gfCNCPoint6[10875] = {X 516.8418, Y 19.7797, Z -8.0000, A 0.000, B 0.000, C 0.000 }
gfCNCPoint6[10876] = {X 516.3652, Y 19.0212, Z -8.0000, A 0.000, B 0.000, C 0.000 }
gfCNCPoint6[10877] = {X 516.0694, Y 18.1758, Z -8.0000, A 0.000, B 0.000, C 0.000 }
gfCNCPoint6[10878] = {X 515.9691, Y 17.2857, Z -8.0000, A 0.000, B 0.000, C 0.000 }
gfCNCPoint6[10879] = {X 515.9691, Y 10.3077, Z -8.0000, A 0.000, B 0.000, C 0.000 }
gfCNCPoint6[10880] = {X 516.0694, Y 9.4176, Z -8.0000, A 0.000, B 0.000, C 0.000 }
gfCNCPoint6[10881] = {X 516.3652, Y 8.5721, Z -8.0000, A 0.000, B 0.000, C 0.000 }
gfCNCPoint6[10882] = {X 516.8418, Y 7.8137, Z -8.0000, A 0.000, B 0.000, C 0.000 }
gfCNCPoint6[10883] = {X 517.4752, Y 7.1803, Z -8.0000, A 0.000, B 0.000, C 0.000 }
gfCNCPoint6[10884] = {X 518.2336, Y 6.7038, Z -8.0000, A 0.000, B 0.000, C 0.000 }
gfCNCPoint6[10885] = {X 519.0791, Y 6.4080, Z -8.0000, A 0.000, B 0.000, C 0.000 }
gfCNCPoint6[10886] = {X 519.9692, Y 6.3077, Z -8.0000, A 0.000, B 0.000, C 0.000 }
gfCNCPoint6[10887] = {X 520.6473, Y 6.3079, Z -8.0000, A 0.000, B 0.000, C 0.000 }
gfCNCPoint6[10888] = {X 521.4439, Y 6.3954, Z -8.0000, A 0.000, B 0.000, C 0.000 }
gfCNCPoint6[10889] = {X 522.2072, Y 6.6401, Z -8.0000, A 0.000, B 0.000, C 0.000 }
gfCNCPoint6[10890] = {X 522.9063, Y 7.0319, Z -8.0000, A 0.000, B 0.000, C 0.000 }
gfCNCPoint6[10891] = {X 523.5133, Y 7.5553, Z -8.0000, A 0.000, B 0.000, C 0.000 }
gfCNCPoint6[10892] = {X 524.0037, Y 8.1892, Z -8.0000, A 0.000, B 0.000, C 0.000 }
gfCNCPoint6[10893] = {X 533.9633, Y 8.1892, Z -8.0000, A 0.000, B 0.000, C 0.000 }
gfCNCPoint6[10894] = {X 533.9633, Y 4.1092, Z -8.0000, A 0.000, B 0.000, C 0.000 }
gfCNCPoint6[10895] = {X 533.9633, Y 4.1092, Z -5.0000, A 0.000, B 0.000, C 0.000 }
gfCNCPoint6[10896] = {X 533.9633, Y 4.1092, Z 11.0000, A 0.000, B 0.000, C 0.000 }
gfCNCPoint6[10897] = {X 419.6152, Y 26.5282, Z 11.0000, A 0.000, B 0.000, C 0.000 }
gfCNCPoint6[10898] = {X 419.6152, Y 26.5282, Z -5.0000, A 0.000, B 0.000, C 0.000 }
gfCNCPoint6[10899] = {X 419.6152, Y 26.5282, Z -8.0000, A 0.000, B 0.000, C 0.000 }
gfCNCPoint6[10900] = {X 416.1517, Y 24.3717, Z -8.0000, A 0.000, B 0.000, C 0.000 }
gfCNCPoint6[10901] = {X 411.5482, Y 31.7655, Z -8.0000, A 0.000, B 0.000, C 0.000 }
gfCNCPoint6[10902] = {X 411.5488, Y 40.8974, Z -8.0000, A 0.000, B 0.000, C 0.000 }
gfCNCPoint6[10903] = {X 412.1870, Y 41.5833, Z -8.0000, A 0.000, B 0.000, C 0.000 }
gfCNCPoint6[10904] = {X 412.6670, Y 42.3878, Z -8.0000, A 0.000, B 0.000, C 0.000 }
gfCNCPoint6[10905] = {X 412.9674, Y 43.2752, Z -8.0000, A 0.000, B 0.000, C 0.000 }
gfCNCPoint6[10906] = {X 413.0747, Y 44.2059, Z -8.0000, A 0.000, B 0.000, C 0.000 }
gfCNCPoint6[10907] = {X 413.0745, Y 45.0415, Z -8.0000, A 0.000, B 0.000, C 0.000 }
gfCNCPoint6[10908] = {X 412.9583, Y 45.9960, Z -8.0000, A 0.000, B 0.000, C 0.000 }
gfCNCPoint6[10909] = {X 412.6339, Y 46.9011, Z -8.0000, A 0.000, B 0.000, C 0.000 }
gfCNCPoint6[10910] = {X 412.1173, Y 47.7120, Z -8.0000, A 0.000, B 0.000, C 0.000 }
gfCNCPoint6[10911] = {X 411.4342, Y 48.3886, Z -8.0000, A 0.000, B 0.000, C 0.000 }
gfCNCPoint6[10912] = {X 410.6184, Y 48.8973, Z -8.0000, A 0.000, B 0.000, C 0.000 }
gfCNCPoint6[10913] = {X 409.7102, Y 49.2130, Z -8.0000, A 0.000, B 0.000, C 0.000 }
gfCNCPoint6[10914] = {X 408.7547, Y 49.3200, Z -8.0000, A 0.000, B 0.000, C 0.000 }
gfCNCPoint6[10915] = {X 402.3112, Y 49.3200, Z -8.0000, A 0.000, B 0.000, C 0.000 }
gfCNCPoint6[10916] = {X 401.3546, Y 49.2127, Z -8.0000, A 0.000, B 0.000, C 0.000 }
gfCNCPoint6[10917] = {X 400.4455, Y 48.8963, Z -8.0000, A 0.000, B 0.000, C 0.000 }
gfCNCPoint6[10918] = {X 399.6290, Y 48.3864, Z -8.0000, A 0.000, B 0.000, C 0.000 }
gfCNCPoint6[10919] = {X 398.9457, Y 47.7084, Z -8.0000, A 0.000, B 0.000, C 0.000 }
gfCNCPoint6[10920] = {X 398.4295, Y 46.8959, Z -8.0000, A 0.000, B 0.000, C 0.000 }
gfCNCPoint6[10921] = {X 398.1060, Y 45.9892, Z -8.0000, A 0.000, B 0.000, C 0.000 }
gfCNCPoint6[10922] = {X 397.9913, Y 45.0335, Z -8.0000, A 0.000, B 0.000, C 0.000 }
gfCNCPoint6[10923] = {X 397.9916, Y 44.1528, Z -8.0000, A 0.000, B 0.000, C 0.000 }
gfCNCPoint6[10924] = {X 398.1015, Y 43.2391, Z -8.0000, A 0.000, B 0.000, C 0.000 }
gfCNCPoint6[10925] = {X 398.4024, Y 42.3694, Z -8.0000, A 0.000, B 0.000, C 0.000 }
gfCNCPoint6[10926] = {X 398.8807, Y 41.5832, Z -8.0000, A 0.000, B 0.000, C 0.000 }
gfCNCPoint6[10927] = {X 399.5147, Y 40.9161, Z -8.0000, A 0.000, B 0.000, C 0.000 }
gfCNCPoint6[10928] = {X 399.4729, Y 31.6029, Z -8.0000, A 0.000, B 0.000, C 0.000 }
gfCNCPoint6[10929] = {X 393.4346, Y 21.1023, Z -8.0000, A 0.000, B 0.000, C 0.000 }
gfCNCPoint6[10930] = {X 392.5863, Y 19.6607, Z -8.0000, A 0.000, B 0.000, C 0.000 }
gfCNCPoint6[10931] = {X 391.7093, Y 18.2363, Z -8.0000, A 0.000, B 0.000, C 0.000 }
gfCNCPoint6[10932] = {X 391.2277, Y 17.5680, Z -8.0000, A 0.000, B 0.000, C 0.000 }
gfCNCPoint6[10933] = {X 390.6666, Y 16.9651, Z -8.0000, A 0.000, B 0.000, C 0.000 }
gfCNCPoint6[10934] = {X 389.7900, Y 16.4727, Z -8.0000, A 0.000, B 0.000, C 0.000 }
gfCNCPoint6[10935] = {X 389.0509, Y 15.7909, Z -8.0000, A 0.000, B 0.000, C 0.000 }
gfCNCPoint6[10936] = {X 388.4895, Y 14.9568, Z -8.0000, A 0.000, B 0.000, C 0.000 }
gfCNCPoint6[10937] = {X 388.1361, Y 14.0155, Z -8.0000, A 0.000, B 0.000, C 0.000 }
gfCNCPoint6[10938] = {X 388.0098, Y 13.0180, Z -8.0000, A 0.000, B 0.000, C 0.000 }
gfCNCPoint6[10939] = {X 388.0096, Y 12.1868, Z -8.0000, A 0.000, B 0.000, C 0.000 }
gfCNCPoint6[10940] = {X 388.1179, Y 11.2255, Z -8.0000, A 0.000, B 0.000, C 0.000 }
gfCNCPoint6[10941] = {X 388.4374, Y 10.3125, Z -8.0000, A 0.000, B 0.000, C 0.000 }
gfCNCPoint6[10942] = {X 388.9521, Y 9.4933, Z -8.0000, A 0.000, B 0.000, C 0.000 }
gfCNCPoint6[10943] = {X 389.6361, Y 8.8093, Z -8.0000, A 0.000, B 0.000, C 0.000 }
gfCNCPoint6[10944] = {X 390.4552, Y 8.2946, Z -8.0000, A 0.000, B 0.000, C 0.000 }
gfCNCPoint6[10945] = {X 391.3683, Y 7.9751, Z -8.0000, A 0.000, B 0.000, C 0.000 }
gfCNCPoint6[10946] = {X 392.3296, Y 7.8668, Z -8.0000, A 0.000, B 0.000, C 0.000 }
gfCNCPoint6[10947] = {X 399.1118, Y 7.8668, Z -8.0000, A 0.000, B 0.000, C 0.000 }
gfCNCPoint6[10948] = {X 400.0730, Y 7.9751, Z -8.0000, A 0.000, B 0.000, C 0.000 }
gfCNCPoint6[10949] = {X 400.9861, Y 8.2946, Z -8.0000, A 0.000, B 0.000, C 0.000 }
gfCNCPoint6[10950] = {X 401.8052, Y 8.8093, Z -8.0000, A 0.000, B 0.000, C 0.000 }
gfCNCPoint6[10951] = {X 402.4893, Y 9.4933, Z -8.0000, A 0.000, B 0.000, C 0.000 }
gfCNCPoint6[10952] = {X 403.0039, Y 10.3124, Z -8.0000, A 0.000, B 0.000, C 0.000 }
gfCNCPoint6[10953] = {X 403.3234, Y 11.2255, Z -8.0000, A 0.000, B 0.000, C 0.000 }
gfCNCPoint6[10954] = {X 403.4318, Y 12.1868, Z -8.0000, A 0.000, B 0.000, C 0.000 }
gfCNCPoint6[10955] = {X 403.4318, Y 12.9782, Z -8.0000, A 0.000, B 0.000, C 0.000 }
gfCNCPoint6[10956] = {X 403.3293, Y 13.9135, Z -8.0000, A 0.000, B 0.000, C 0.000 }
gfCNCPoint6[10957] = {X 403.0267, Y 14.8044, Z -8.0000, A 0.000, B 0.000, C 0.000 }
gfCNCPoint6[10958] = {X 405.3554, Y 18.8222, Z -8.0000, A 0.000, B 0.000, C 0.000 }
gfCNCPoint6[10959] = {X 407.8730, Y 14.7530, Z -8.0000, A 0.000, B 0.000, C 0.000 }
gfCNCPoint6[10960] = {X 407.5919, Y 13.9039, Z -8.0000, A 0.000, B 0.000, C 0.000 }
gfCNCPoint6[10961] = {X 407.4917, Y 13.0151, Z -8.0000, A 0.000, B 0.000, C 0.000 }
gfCNCPoint6[10962] = {X 407.4915, Y 12.1868, Z -8.0000, A 0.000, B 0.000, C 0.000 }
gfCNCPoint6[10963] = {X 407.5999, Y 11.2255, Z -8.0000, A 0.000, B 0.000, C 0.000 }
gfCNCPoint6[10964] = {X 407.9194, Y 10.3124, Z -8.0000, A 0.000, B 0.000, C 0.000 }
gfCNCPoint6[10965] = {X 408.4340, Y 9.4933, Z -8.0000, A 0.000, B 0.000, C 0.000 }
gfCNCPoint6[10966] = {X 409.1181, Y 8.8093, Z -8.0000, A 0.000, B 0.000, C 0.000 }
gfCNCPoint6[10967] = {X 409.9372, Y 8.2946, Z -8.0000, A 0.000, B 0.000, C 0.000 }
gfCNCPoint6[10968] = {X 410.8502, Y 7.9751, Z -8.0000, A 0.000, B 0.000, C 0.000 }
gfCNCPoint6[10969] = {X 411.8115, Y 7.8668, Z -8.0000, A 0.000, B 0.000, C 0.000 }
gfCNCPoint6[10970] = {X 419.3245, Y 7.8668, Z -8.0000, A 0.000, B 0.000, C 0.000 }
gfCNCPoint6[10971] = {X 420.2858, Y 7.9751, Z -8.0000, A 0.000, B 0.000, C 0.000 }
gfCNCPoint6[10972] = {X 421.1988, Y 8.2946, Z -8.0000, A 0.000, B 0.000, C 0.000 }
gfCNCPoint6[10973] = {X 422.0179, Y 8.8093, Z -8.0000, A 0.000, B 0.000, C 0.000 }
gfCNCPoint6[10974] = {X 422.7020, Y 9.4933, Z -8.0000, A 0.000, B 0.000, C 0.000 }
gfCNCPoint6[10975] = {X 423.2166, Y 10.3124, Z -8.0000, A 0.000, B 0.000, C 0.000 }
gfCNCPoint6[10976] = {X 423.5361, Y 11.2255, Z -8.0000, A 0.000, B 0.000, C 0.000 }
gfCNCPoint6[10977] = {X 423.6445, Y 12.1868, Z -8.0000, A 0.000, B 0.000, C 0.000 }
gfCNCPoint6[10978] = {X 423.6445, Y 12.9801, Z -8.0000, A 0.000, B 0.000, C 0.000 }
gfCNCPoint6[10979] = {X 423.5522, Y 13.8467, Z -8.0000, A 0.000, B 0.000, C 0.000 }
gfCNCPoint6[10980] = {X 423.2901, Y 14.6779, Z -8.0000, A 0.000, B 0.000, C 0.000 }
gfCNCPoint6[10981] = {X 422.8686, Y 15.4407, Z -8.0000, A 0.000, B 0.000, C 0.000 }
gfCNCPoint6[10982] = {X 422.3045, Y 16.1050, Z -8.0000, A 0.000, B 0.000, C 0.000 }
gfCNCPoint6[10983] = {X 421.6199, Y 16.6444, Z -8.0000, A 0.000, B 0.000, C 0.000 }
gfCNCPoint6[10984] = {X 420.8421, Y 17.0376, Z -8.0000, A 0.000, B 0.000, C 0.000 }
gfCNCPoint6[10985] = {X 420.1257, Y 18.0009, Z -8.0000, A 0.000, B 0.000, C 0.000 }
gfCNCPoint6[10986] = {X 419.4776, Y 19.0115, Z -8.0000, A 0.000, B 0.000, C 0.000 }
gfCNCPoint6[10987] = {X 417.9942, Y 21.4124, Z -8.0000, A 0.000, B 0.000, C 0.000 }
gfCNCPoint6[10988] = {X 416.1517, Y 24.3717, Z -8.0000, A 0.000, B 0.000, C 0.000 }
gfCNCPoint6[10989] = {X 419.5473, Y 26.4859, Z -8.0000, A 0.000, B 0.000, C 0.000 }
gfCNCPoint6[10990] = {X 416.0838, Y 24.3294, Z -8.0000, A 0.000, B 0.000, C 0.000 }
gfCNCPoint6[10991] = {X 411.4682, Y 31.7426, Z -8.0000, A 0.000, B 0.000, C 0.000 }
gfCNCPoint6[10992] = {X 411.4688, Y 40.9341, Z -8.0000, A 0.000, B 0.000, C 0.000 }
gfCNCPoint6[10993] = {X 412.1066, Y 41.6095, Z -8.0000, A 0.000, B 0.000, C 0.000 }
gfCNCPoint6[10994] = {X 412.5867, Y 42.4049, Z -8.0000, A 0.000, B 0.000, C 0.000 }
gfCNCPoint6[10995] = {X 412.8873, Y 43.2839, Z -8.0000, A 0.000, B 0.000, C 0.000 }
gfCNCPoint6[10996] = {X 412.9947, Y 44.2067, Z -8.0000, A 0.000, B 0.000, C 0.000 }
gfCNCPoint6[10997] = {X 412.9945, Y 45.0408, Z -8.0000, A 0.000, B 0.000, C 0.000 }
gfCNCPoint6[10998] = {X 412.8805, Y 45.9775, Z -8.0000, A 0.000, B 0.000, C 0.000 }
gfCNCPoint6[10999] = {X 412.5621, Y 46.8659, Z -8.0000, A 0.000, B 0.000, C 0.000 }
gfCNCPoint6[11000] = {X 412.0551, Y 47.6618, Z -8.0000, A 0.000, B 0.000, C 0.000 }
gfCNCPoint6[11001] = {X 411.3846, Y 48.3258, Z -8.0000, A 0.000, B 0.000, C 0.000 }
gfCNCPoint6[11002] = {X 410.5838, Y 48.8251, Z -8.0000, A 0.000, B 0.000, C 0.000 }
gfCNCPoint6[11003] = {X 409.6925, Y 49.1350, Z -8.0000, A 0.000, B 0.000, C 0.000 }
gfCNCPoint6[11004] = {X 408.7547, Y 49.2400, Z -8.0000, A 0.000, B 0.000, C 0.000 }
gfCNCPoint6[11005] = {X 402.3112, Y 49.2400, Z -8.0000, A 0.000, B 0.000, C 0.000 }
gfCNCPoint6[11006] = {X 401.3723, Y 49.1347, Z -8.0000, A 0.000, B 0.000, C 0.000 }
gfCNCPoint6[11007] = {X 400.4800, Y 48.8242, Z -8.0000, A 0.000, B 0.000, C 0.000 }
gfCNCPoint6[11008] = {X 399.6786, Y 48.3237, Z -8.0000, A 0.000, B 0.000, C 0.000 }
gfCNCPoint6[11009] = {X 399.0080, Y 47.6582, Z -8.0000, A 0.000, B 0.000, C 0.000 }
gfCNCPoint6[11010] = {X 398.5013, Y 46.8608, Z -8.0000, A 0.000, B 0.000, C 0.000 }
gfCNCPoint6[11011] = {X 398.1839, Y 45.9709, Z -8.0000, A 0.000, B 0.000, C 0.000 }
gfCNCPoint6[11012] = {X 398.0713, Y 45.0329, Z -8.0000, A 0.000, B 0.000, C 0.000 }
gfCNCPoint6[11013] = {X 398.0716, Y 44.1538, Z -8.0000, A 0.000, B 0.000, C 0.000 }
gfCNCPoint6[11014] = {X 398.1815, Y 43.2480, Z -8.0000, A 0.000, B 0.000, C 0.000 }
gfCNCPoint6[11015] = {X 398.4827, Y 42.3867, Z -8.0000, A 0.000, B 0.000, C 0.000 }
gfCNCPoint6[11016] = {X 398.9612, Y 41.6098, Z -8.0000, A 0.000, B 0.000, C 0.000 }
gfCNCPoint6[11017] = {X 399.5948, Y 40.9532, Z -8.0000, A 0.000, B 0.000, C 0.000 }
gfCNCPoint6[11018] = {X 399.5528, Y 31.5814, Z -8.0000, A 0.000, B 0.000, C 0.000 }
gfCNCPoint6[11019] = {X 393.5040, Y 21.0625, Z -8.0000, A 0.000, B 0.000, C 0.000 }
gfCNCPoint6[11020] = {X 392.6548, Y 19.6194, Z -8.0000, A 0.000, B 0.000, C 0.000 }
gfCNCPoint6[11021] = {X 391.7770, Y 18.1936, Z -8.0000, A 0.000, B 0.000, C 0.000 }
gfCNCPoint6[11022] = {X 391.2849, Y 17.5116, Z -8.0000, A 0.000, B 0.000, C 0.000 }
gfCNCPoint6[11023] = {X 390.7109, Y 16.8969, Z -8.0000, A 0.000, B 0.000, C 0.000 }
gfCNCPoint6[11024] = {X 389.8465, Y 16.4148, Z -8.0000, A 0.000, B 0.000, C 0.000 }
gfCNCPoint6[11025] = {X 389.1174, Y 15.7455, Z -8.0000, A 0.000, B 0.000, C 0.000 }
gfCNCPoint6[11026] = {X 388.5633, Y 14.9254, Z -8.0000, A 0.000, B 0.000, C 0.000 }
gfCNCPoint6[11027] = {X 388.2144, Y 13.9992, Z -8.0000, A 0.000, B 0.000, C 0.000 }
gfCNCPoint6[11028] = {X 388.0898, Y 13.0173, Z -8.0000, A 0.000, B 0.000, C 0.000 }
gfCNCPoint6[11029] = {X 388.0896, Y 12.1868, Z -8.0000, A 0.000, B 0.000, C 0.000 }
gfCNCPoint6[11030] = {X 388.1959, Y 11.2433, Z -8.0000, A 0.000, B 0.000, C 0.000 }
gfCNCPoint6[11031] = {X 388.5095, Y 10.3472, Z -8.0000, A 0.000, B 0.000, C 0.000 }
gfCNCPoint6[11032] = {X 389.0147, Y 9.5432, Z -8.0000, A 0.000, B 0.000, C 0.000 }
gfCNCPoint6[11033] = {X 389.6860, Y 8.8719, Z -8.0000, A 0.000, B 0.000, C 0.000 }
gfCNCPoint6[11034] = {X 390.4900, Y 8.3667, Z -8.0000, A 0.000, B 0.000, C 0.000 }
gfCNCPoint6[11035] = {X 391.3861, Y 8.0531, Z -8.0000, A 0.000, B 0.000, C 0.000 }
gfCNCPoint6[11036] = {X 392.3296, Y 7.9468, Z -8.0000, A 0.000, B 0.000, C 0.000 }
gfCNCPoint6[11037] = {X 399.1118, Y 7.9468, Z -8.0000, A 0.000, B 0.000, C 0.000 }
gfCNCPoint6[11038] = {X 400.0552, Y 8.0531, Z -8.0000, A 0.000, B 0.000, C 0.000 }
gfCNCPoint6[11039] = {X 400.9514, Y 8.3667, Z -8.0000, A 0.000, B 0.000, C 0.000 }
gfCNCPoint6[11040] = {X 401.7554, Y 8.8718, Z -8.0000, A 0.000, B 0.000, C 0.000 }
gfCNCPoint6[11041] = {X 402.4267, Y 9.5432, Z -8.0000, A 0.000, B 0.000, C 0.000 }
gfCNCPoint6[11042] = {X 402.9319, Y 10.3471, Z -8.0000, A 0.000, B 0.000, C 0.000 }
gfCNCPoint6[11043] = {X 403.2455, Y 11.2433, Z -8.0000, A 0.000, B 0.000, C 0.000 }
gfCNCPoint6[11044] = {X 403.3518, Y 12.1868, Z -8.0000, A 0.000, B 0.000, C 0.000 }
gfCNCPoint6[11045] = {X 403.3518, Y 12.9782, Z -8.0000, A 0.000, B 0.000, C 0.000 }
gfCNCPoint6[11046] = {X 403.2466, Y 13.9164, Z -8.0000, A 0.000, B 0.000, C 0.000 }
gfCNCPoint6[11047] = {X 402.9364, Y 14.8081, Z -8.0000, A 0.000, B 0.000, C 0.000 }
gfCNCPoint6[11048] = {X 405.3532, Y 18.9779, Z -8.0000, A 0.000, B 0.000, C 0.000 }
gfCNCPoint6[11049] = {X 407.9636, Y 14.7587, Z -8.0000, A 0.000, B 0.000, C 0.000 }
gfCNCPoint6[11050] = {X 407.6747, Y 13.9075, Z -8.0000, A 0.000, B 0.000, C 0.000 }
gfCNCPoint6[11051] = {X 407.5717, Y 13.0144, Z -8.0000, A 0.000, B 0.000, C 0.000 }
gfCNCPoint6[11052] = {X 407.5715, Y 12.1868, Z -8.0000, A 0.000, B 0.000, C 0.000 }
gfCNCPoint6[11053] = {X 407.6778, Y 11.2433, Z -8.0000, A 0.000, B 0.000, C 0.000 }
gfCNCPoint6[11054] = {X 407.9914, Y 10.3471, Z -8.0000, A 0.000, B 0.000, C 0.000 }
gfCNCPoint6[11055] = {X 408.4966, Y 9.5432, Z -8.0000, A 0.000, B 0.000, C 0.000 }
gfCNCPoint6[11056] = {X 409.1679, Y 8.8718, Z -8.0000, A 0.000, B 0.000, C 0.000 }
gfCNCPoint6[11057] = {X 409.9719, Y 8.3667, Z -8.0000, A 0.000, B 0.000, C 0.000 }
gfCNCPoint6[11058] = {X 410.8681, Y 8.0531, Z -8.0000, A 0.000, B 0.000, C 0.000 }
gfCNCPoint6[11059] = {X 411.8115, Y 7.9468, Z -8.0000, A 0.000, B 0.000, C 0.000 }
gfCNCPoint6[11060] = {X 419.3245, Y 7.9468, Z -8.0000, A 0.000, B 0.000, C 0.000 }
gfCNCPoint6[11061] = {X 420.2679, Y 8.0531, Z -8.0000, A 0.000, B 0.000, C 0.000 }
gfCNCPoint6[11062] = {X 421.1641, Y 8.3667, Z -8.0000, A 0.000, B 0.000, C 0.000 }
gfCNCPoint6[11063] = {X 421.9681, Y 8.8718, Z -8.0000, A 0.000, B 0.000, C 0.000 }
gfCNCPoint6[11064] = {X 422.6394, Y 9.5432, Z -8.0000, A 0.000, B 0.000, C 0.000 }
gfCNCPoint6[11065] = {X 423.1446, Y 10.3471, Z -8.0000, A 0.000, B 0.000, C 0.000 }
gfCNCPoint6[11066] = {X 423.4582, Y 11.2433, Z -8.0000, A 0.000, B 0.000, C 0.000 }
gfCNCPoint6[11067] = {X 423.5645, Y 12.1868, Z -8.0000, A 0.000, B 0.000, C 0.000 }
gfCNCPoint6[11068] = {X 423.5645, Y 12.9795, Z -8.0000, A 0.000, B 0.000, C 0.000 }
gfCNCPoint6[11069] = {X 423.4731, Y 13.8339, Z -8.0000, A 0.000, B 0.000, C 0.000 }
gfCNCPoint6[11070] = {X 423.2137, Y 14.6529, Z -8.0000, A 0.000, B 0.000, C 0.000 }
gfCNCPoint6[11071] = {X 422.7967, Y 15.4041, Z -8.0000, A 0.000, B 0.000, C 0.000 }
gfCNCPoint6[11072] = {X 422.2386, Y 16.0574, Z -8.0000, A 0.000, B 0.000, C 0.000 }
gfCNCPoint6[11073] = {X 421.5618, Y 16.5866, Z -8.0000, A 0.000, B 0.000, C 0.000 }
gfCNCPoint6[11074] = {X 420.7932, Y 16.9707, Z -8.0000, A 0.000, B 0.000, C 0.000 }
gfCNCPoint6[11075] = {X 420.0662, Y 17.9462, Z -8.0000, A 0.000, B 0.000, C 0.000 }
gfCNCPoint6[11076] = {X 419.4091, Y 18.9700, Z -8.0000, A 0.000, B 0.000, C 0.000 }
gfCNCPoint6[11077] = {X 417.9262, Y 21.3702, Z -8.0000, A 0.000, B 0.000, C 0.000 }
gfCNCPoint6[11078] = {X 416.0838, Y 24.3294, Z -8.0000, A 0.000, B 0.000, C 0.000 }
gfCNCPoint6[11079] = {X 419.4794, Y 26.4436, Z -8.0000, A 0.000, B 0.000, C 0.000 }
gfCNCPoint6[11080] = {X 416.0159, Y 24.2871, Z -8.0000, A 0.000, B 0.000, C 0.000 }
gfCNCPoint6[11081] = {X 411.3882, Y 31.7197, Z -8.0000, A 0.000, B 0.000, C 0.000 }
gfCNCPoint6[11082] = {X 411.3888, Y 40.9711, Z -8.0000, A 0.000, B 0.000, C 0.000 }
gfCNCPoint6[11083] = {X 412.0262, Y 41.6361, Z -8.0000, A 0.000, B 0.000, C 0.000 }
gfCNCPoint6[11084] = {X 412.5064, Y 42.4220, Z -8.0000, A 0.000, B 0.000, C 0.000 }
gfCNCPoint6[11085] = {X 412.8072, Y 43.2926, Z -8.0000, A 0.000, B 0.000, C 0.000 }
gfCNCPoint6[11086] = {X 412.9147, Y 44.2074, Z -8.0000, A 0.000, B 0.000, C 0.000 }
gfCNCPoint6[11087] = {X 412.9145, Y 45.0400, Z -8.0000, A 0.000, B 0.000, C 0.000 }
gfCNCPoint6[11088] = {X 412.8026, Y 45.9591, Z -8.0000, A 0.000, B 0.000, C 0.000 }
gfCNCPoint6[11089] = {X 412.4902, Y 46.8306, Z -8.0000, A 0.000, B 0.000, C 0.000 }
gfCNCPoint6[11090] = {X 411.9928, Y 47.6115, Z -8.0000, A 0.000, B 0.000, C 0.000 }
gfCNCPoint6[11091] = {X 411.3350, Y 48.2631, Z -8.0000, A 0.000, B 0.000, C 0.000 }
gfCNCPoint6[11092] = {X 410.5493, Y 48.7530, Z -8.0000, A 0.000, B 0.000, C 0.000 }
gfCNCPoint6[11093] = {X 409.6748, Y 49.0570, Z -8.0000, A 0.000, B 0.000, C 0.000 }
gfCNCPoint6[11094] = {X 408.7547, Y 49.1600, Z -8.0000, A 0.000, B 0.000, C 0.000 }
gfCNCPoint6[11095] = {X 402.3112, Y 49.1600, Z -8.0000, A 0.000, B 0.000, C 0.000 }
gfCNCPoint6[11096] = {X 401.3900, Y 49.0567, Z -8.0000, A 0.000, B 0.000, C 0.000 }
gfCNCPoint6[11097] = {X 400.5146, Y 48.7520, Z -8.0000, A 0.000, B 0.000, C 0.000 }
gfCNCPoint6[11098] = {X 399.7283, Y 48.2610, Z -8.0000, A 0.000, B 0.000, C 0.000 }
gfCNCPoint6[11099] = {X 399.0703, Y 47.6081, Z -8.0000, A 0.000, B 0.000, C 0.000 }
gfCNCPoint6[11100] = {X 398.5732, Y 46.8257, Z -8.0000, A 0.000, B 0.000, C 0.000 }
gfCNCPoint6[11101] = {X 398.2617, Y 45.9526, Z -8.0000, A 0.000, B 0.000, C 0.000 }
gfCNCPoint6[11102] = {X 398.1513, Y 45.0322, Z -8.0000, A 0.000, B 0.000, C 0.000 }
gfCNCPoint6[11103] = {X 398.1516, Y 44.1549, Z -8.0000, A 0.000, B 0.000, C 0.000 }
gfCNCPoint6[11104] = {X 398.2616, Y 43.2570, Z -8.0000, A 0.000, B 0.000, C 0.000 }
gfCNCPoint6[11105] = {X 398.5630, Y 42.4041, Z -8.0000, A 0.000, B 0.000, C 0.000 }
gfCNCPoint6[11106] = {X 399.0417, Y 41.6366, Z -8.0000, A 0.000, B 0.000, C 0.000 }
gfCNCPoint6[11107] = {X 399.6750, Y 40.9907, Z -8.0000, A 0.000, B 0.000, C 0.000 }
gfCNCPoint6[11108] = {X 399.6327, Y 31.5599, Z -8.0000, A 0.000, B 0.000, C 0.000 }
gfCNCPoint6[11109] = {X 393.5733, Y 21.0226, Z -8.0000, A 0.000, B 0.000, C 0.000 }
gfCNCPoint6[11110] = {X 392.7234, Y 19.5782, Z -8.0000, A 0.000, B 0.000, C 0.000 }
gfCNCPoint6[11111] = {X 391.8447, Y 18.1510, Z -8.0000, A 0.000, B 0.000, C 0.000 }
gfCNCPoint6[11112] = {X 391.3420, Y 17.4550, Z -8.0000, A 0.000, B 0.000, C 0.000 }
gfCNCPoint6[11113] = {X 390.7550, Y 16.8285, Z -8.0000, A 0.000, B 0.000, C 0.000 }
gfCNCPoint6[11114] = {X 389.9028, Y 16.3568, Z -8.0000, A 0.000, B 0.000, C 0.000 }
gfCNCPoint6[11115] = {X 389.1837, Y 15.6999, Z -8.0000, A 0.000, B 0.000, C 0.000 }
gfCNCPoint6[11116] = {X 388.6370, Y 14.8938, Z -8.0000, A 0.000, B 0.000, C 0.000 }
gfCNCPoint6[11117] = {X 388.2928, Y 13.9827, Z -8.0000, A 0.000, B 0.000, C 0.000 }
gfCNCPoint6[11118] = {X 388.1698, Y 13.0166, Z -8.0000, A 0.000, B 0.000, C 0.000 }
gfCNCPoint6[11119] = {X 388.1696, Y 12.1868, Z -8.0000, A 0.000, B 0.000, C 0.000 }
gfCNCPoint6[11120] = {X 388.2739, Y 11.2611, Z -8.0000, A 0.000, B 0.000, C 0.000 }
gfCNCPoint6[11121] = {X 388.5816, Y 10.3819, Z -8.0000, A 0.000, B 0.000, C 0.000 }
gfCNCPoint6[11122] = {X 389.0772, Y 9.5931, Z -8.0000, A 0.000, B 0.000, C 0.000 }
gfCNCPoint6[11123] = {X 389.7359, Y 8.9344, Z -8.0000, A 0.000, B 0.000, C 0.000 }
gfCNCPoint6[11124] = {X 390.5247, Y 8.4388, Z -8.0000, A 0.000, B 0.000, C 0.000 }
gfCNCPoint6[11125] = {X 391.4039, Y 8.1311, Z -8.0000, A 0.000, B 0.000, C 0.000 }
gfCNCPoint6[11126] = {X 392.3296, Y 8.0268, Z -8.0000, A 0.000, B 0.000, C 0.000 }
gfCNCPoint6[11127] = {X 399.1118, Y 8.0268, Z -8.0000, A 0.000, B 0.000, C 0.000 }
gfCNCPoint6[11128] = {X 400.0374, Y 8.1311, Z -8.0000, A 0.000, B 0.000, C 0.000 }
gfCNCPoint6[11129] = {X 400.9167, Y 8.4388, Z -8.0000, A 0.000, B 0.000, C 0.000 }
gfCNCPoint6[11130] = {X 401.7055, Y 8.9344, Z -8.0000, A 0.000, B 0.000, C 0.000 }
gfCNCPoint6[11131] = {X 402.3642, Y 9.5931, Z -8.0000, A 0.000, B 0.000, C 0.000 }
gfCNCPoint6[11132] = {X 402.8598, Y 10.3819, Z -8.0000, A 0.000, B 0.000, C 0.000 }
gfCNCPoint6[11133] = {X 403.1675, Y 11.2611, Z -8.0000, A 0.000, B 0.000, C 0.000 }
gfCNCPoint6[11134] = {X 403.2718, Y 12.1868, Z -8.0000, A 0.000, B 0.000, C 0.000 }
gfCNCPoint6[11135] = {X 403.2718, Y 12.9782, Z -8.0000, A 0.000, B 0.000, C 0.000 }
gfCNCPoint6[11136] = {X 403.1639, Y 13.9192, Z -8.0000, A 0.000, B 0.000, C 0.000 }
gfCNCPoint6[11137] = {X 402.8459, Y 14.8115, Z -8.0000, A 0.000, B 0.000, C 0.000 }
gfCNCPoint6[11138] = {X 405.3509, Y 19.1335, Z -8.0000, A 0.000, B 0.000, C 0.000 }
gfCNCPoint6[11139] = {X 408.0544, Y 14.7640, Z -8.0000, A 0.000, B 0.000, C 0.000 }
gfCNCPoint6[11140] = {X 407.7575, Y 13.9109, Z -8.0000, A 0.000, B 0.000, C 0.000 }
gfCNCPoint6[11141] = {X 407.6517, Y 13.0137, Z -8.0000, A 0.000, B 0.000, C 0.000 }
gfCNCPoint6[11142] = {X 407.6515, Y 12.1868, Z -8.0000, A 0.000, B 0.000, C 0.000 }
gfCNCPoint6[11143] = {X 407.7558, Y 11.2611, Z -8.0000, A 0.000, B 0.000, C 0.000 }
gfCNCPoint6[11144] = {X 408.0635, Y 10.3819, Z -8.0000, A 0.000, B 0.000, C 0.000 }
gfCNCPoint6[11145] = {X 408.5591, Y 9.5931, Z -8.0000, A 0.000, B 0.000, C 0.000 }
gfCNCPoint6[11146] = {X 409.2178, Y 8.9344, Z -8.0000, A 0.000, B 0.000, C 0.000 }
gfCNCPoint6[11147] = {X 410.0066, Y 8.4388, Z -8.0000, A 0.000, B 0.000, C 0.000 }
gfCNCPoint6[11148] = {X 410.8859, Y 8.1311, Z -8.0000, A 0.000, B 0.000, C 0.000 }
gfCNCPoint6[11149] = {X 411.8115, Y 8.0268, Z -8.0000, A 0.000, B 0.000, C 0.000 }
gfCNCPoint6[11150] = {X 419.3245, Y 8.0268, Z -8.0000, A 0.000, B 0.000, C 0.000 }
gfCNCPoint6[11151] = {X 420.2501, Y 8.1311, Z -8.0000, A 0.000, B 0.000, C 0.000 }
gfCNCPoint6[11152] = {X 421.1294, Y 8.4388, Z -8.0000, A 0.000, B 0.000, C 0.000 }
gfCNCPoint6[11153] = {X 421.9182, Y 8.9344, Z -8.0000, A 0.000, B 0.000, C 0.000 }
gfCNCPoint6[11154] = {X 422.5769, Y 9.5931, Z -8.0000, A 0.000, B 0.000, C 0.000 }
gfCNCPoint6[11155] = {X 423.0725, Y 10.3819, Z -8.0000, A 0.000, B 0.000, C 0.000 }
gfCNCPoint6[11156] = {X 423.3802, Y 11.2611, Z -8.0000, A 0.000, B 0.000, C 0.000 }
gfCNCPoint6[11157] = {X 423.4845, Y 12.1868, Z -8.0000, A 0.000, B 0.000, C 0.000 }
gfCNCPoint6[11158] = {X 423.4845, Y 12.9790, Z -8.0000, A 0.000, B 0.000, C 0.000 }
gfCNCPoint6[11159] = {X 423.3941, Y 13.8210, Z -8.0000, A 0.000, B 0.000, C 0.000 }
gfCNCPoint6[11160] = {X 423.1374, Y 14.6279, Z -8.0000, A 0.000, B 0.000, C 0.000 }
gfCNCPoint6[11161] = {X 422.7248, Y 15.3674, Z -8.0000, A 0.000, B 0.000, C 0.000 }
gfCNCPoint6[11162] = {X 422.1728, Y 16.0096, Z -8.0000, A 0.000, B 0.000, C 0.000 }
gfCNCPoint6[11163] = {X 421.5037, Y 16.5286, Z -8.0000, A 0.000, B 0.000, C 0.000 }
gfCNCPoint6[11164] = {X 420.7445, Y 16.9036, Z -8.0000, A 0.000, B 0.000, C 0.000 }
gfCNCPoint6[11165] = {X 420.0069, Y 17.8913, Z -8.0000, A 0.000, B 0.000, C 0.000 }
gfCNCPoint6[11166] = {X 419.3407, Y 18.9286, Z -8.0000, A 0.000, B 0.000, C 0.000 }
gfCNCPoint6[11167] = {X 417.8582, Y 21.3280, Z -8.0000, A 0.000, B 0.000, C 0.000 }
gfCNCPoint6[11168] = {X 416.0159, Y 24.2871, Z -8.0000, A 0.000, B 0.000, C 0.000 }
gfCNCPoint6[11169] = {X 419.4115, Y 26.4013, Z -8.0000, A 0.000, B 0.000, C 0.000 }
gfCNCPoint6[11170] = {X 415.9479, Y 24.2449, Z -8.0000, A 0.000, B 0.000, C 0.000 }
gfCNCPoint6[11171] = {X 411.3082, Y 31.6969, Z -8.0000, A 0.000, B 0.000, C 0.000 }
gfCNCPoint6[11172] = {X 411.3088, Y 41.0086, Z -8.0000, A 0.000, B 0.000, C 0.000 }
gfCNCPoint6[11173] = {X 411.9457, Y 41.6629, Z -8.0000, A 0.000, B 0.000, C 0.000 }
gfCNCPoint6[11174] = {X 412.4261, Y 42.4394, Z -8.0000, A 0.000, B 0.000, C 0.000 }
gfCNCPoint6[11175] = {X 412.7272, Y 43.3014, Z -8.0000, A 0.000, B 0.000, C 0.000 }
gfCNCPoint6[11176] = {X 412.8347, Y 44.2081, Z -8.0000, A 0.000, B 0.000, C 0.000 }
gfCNCPoint6[11177] = {X 412.8345, Y 45.0392, Z -8.0000, A 0.000, B 0.000, C 0.000 }
gfCNCPoint6[11178] = {X 412.7248, Y 45.9406, Z -8.0000, A 0.000, B 0.000, C 0.000 }
gfCNCPoint6[11179] = {X 412.4184, Y 46.7954, Z -8.0000, A 0.000, B 0.000, C 0.000 }
gfCNCPoint6[11180] = {X 411.9305, Y 47.5613, Z -8.0000, A 0.000, B 0.000, C 0.000 }
gfCNCPoint6[11181] = {X 411.2854, Y 48.2003, Z -8.0000, A 0.000, B 0.000, C 0.000 }
gfCNCPoint6[11182] = {X 410.5148, Y 48.6808, Z -8.0000, A 0.000, B 0.000, C 0.000 }
gfCNCPoint6[11183] = {X 409.6571, Y 48.9789, Z -8.0000, A 0.000, B 0.000, C 0.000 }
gfCNCPoint6[11184] = {X 408.7547, Y 49.0800, Z -8.0000, A 0.000, B 0.000, C 0.000 }
gfCNCPoint6[11185] = {X 402.3112, Y 49.0800, Z -8.0000, A 0.000, B 0.000, C 0.000 }
gfCNCPoint6[11186] = {X 401.4077, Y 48.9787, Z -8.0000, A 0.000, B 0.000, C 0.000 }
gfCNCPoint6[11187] = {X 400.5491, Y 48.6799, Z -8.0000, A 0.000, B 0.000, C 0.000 }
gfCNCPoint6[11188] = {X 399.7780, Y 48.1983, Z -8.0000, A 0.000, B 0.000, C 0.000 }
gfCNCPoint6[11189] = {X 399.1326, Y 47.5579, Z -8.0000, A 0.000, B 0.000, C 0.000 }
gfCNCPoint6[11190] = {X 398.6451, Y 46.7906, Z -8.0000, A 0.000, B 0.000, C 0.000 }
gfCNCPoint6[11191] = {X 398.3396, Y 45.9343, Z -8.0000, A 0.000, B 0.000, C 0.000 }
gfCNCPoint6[11192] = {X 398.2313, Y 45.0316, Z -8.0000, A 0.000, B 0.000, C 0.000 }
gfCNCPoint6[11193] = {X 398.2316, Y 44.1559, Z -8.0000, A 0.000, B 0.000, C 0.000 }
gfCNCPoint6[11194] = {X 398.3416, Y 43.2661, Z -8.0000, A 0.000, B 0.000, C 0.000 }
gfCNCPoint6[11195] = {X 398.6434, Y 42.4218, Z -8.0000, A 0.000, B 0.000, C 0.000 }
gfCNCPoint6[11196] = {X 399.1223, Y 41.6638, Z -8.0000, A 0.000, B 0.000, C 0.000 }
gfCNCPoint6[11197] = {X 399.7552, Y 41.0287, Z -8.0000, A 0.000, B 0.000, C 0.000 }
gfCNCPoint6[11198] = {X 399.7126, Y 31.5384, Z -8.0000, A 0.000, B 0.000, C 0.000 }
gfCNCPoint6[11199] = {X 393.6427, Y 20.9827, Z -8.0000, A 0.000, B 0.000, C 0.000 }
gfCNCPoint6[11200] = {X 392.7919, Y 19.5369, Z -8.0000, A 0.000, B 0.000, C 0.000 }
gfCNCPoint6[11201] = {X 391.9124, Y 18.1084, Z -8.0000, A 0.000, B 0.000, C 0.000 }
gfCNCPoint6[11202] = {X 391.3990, Y 17.3984, Z -8.0000, A 0.000, B 0.000, C 0.000 }
gfCNCPoint6[11203] = {X 390.7989, Y 16.7600, Z -8.0000, A 0.000, B 0.000, C 0.000 }
gfCNCPoint6[11204] = {X 389.9591, Y 16.2987, Z -8.0000, A 0.000, B 0.000, C 0.000 }
gfCNCPoint6[11205] = {X 389.2500, Y 15.6542, Z -8.0000, A 0.000, B 0.000, C 0.000 }
gfCNCPoint6[11206] = {X 388.7108, Y 14.8622, Z -8.0000, A 0.000, B 0.000, C 0.000 }
gfCNCPoint6[11207] = {X 388.3711, Y 13.9663, Z -8.0000, A 0.000, B 0.000, C 0.000 }
gfCNCPoint6[11208] = {X 388.2498, Y 13.0158, Z -8.0000, A 0.000, B 0.000, C 0.000 }
gfCNCPoint6[11209] = {X 388.2496, Y 12.1868, Z -8.0000, A 0.000, B 0.000, C 0.000 }
gfCNCPoint6[11210] = {X 388.3519, Y 11.2789, Z -8.0000, A 0.000, B 0.000, C 0.000 }
gfCNCPoint6[11211] = {X 388.6537, Y 10.4166, Z -8.0000, A 0.000, B 0.000, C 0.000 }
gfCNCPoint6[11212] = {X 389.1398, Y 9.6430, Z -8.0000, A 0.000, B 0.000, C 0.000 }
gfCNCPoint6[11213] = {X 389.7858, Y 8.9969, Z -8.0000, A 0.000, B 0.000, C 0.000 }
gfCNCPoint6[11214] = {X 390.5594, Y 8.5109, Z -8.0000, A 0.000, B 0.000, C 0.000 }
gfCNCPoint6[11215] = {X 391.4217, Y 8.2091, Z -8.0000, A 0.000, B 0.000, C 0.000 }
gfCNCPoint6[11216] = {X 392.3296, Y 8.1068, Z -8.0000, A 0.000, B 0.000, C 0.000 }
gfCNCPoint6[11217] = {X 399.1118, Y 8.1068, Z -8.0000, A 0.000, B 0.000, C 0.000 }
gfCNCPoint6[11218] = {X 400.0196, Y 8.2091, Z -8.0000, A 0.000, B 0.000, C 0.000 }
gfCNCPoint6[11219] = {X 400.8820, Y 8.5109, Z -8.0000, A 0.000, B 0.000, C 0.000 }
gfCNCPoint6[11220] = {X 401.6556, Y 8.9969, Z -8.0000, A 0.000, B 0.000, C 0.000 }
gfCNCPoint6[11221] = {X 402.3016, Y 9.6430, Z -8.0000, A 0.000, B 0.000, C 0.000 }
gfCNCPoint6[11222] = {X 402.7877, Y 10.4166, Z -8.0000, A 0.000, B 0.000, C 0.000 }
gfCNCPoint6[11223] = {X 403.0895, Y 11.2789, Z -8.0000, A 0.000, B 0.000, C 0.000 }
gfCNCPoint6[11224] = {X 403.1918, Y 12.1868, Z -8.0000, A 0.000, B 0.000, C 0.000 }
gfCNCPoint6[11225] = {X 403.1918, Y 12.9782, Z -8.0000, A 0.000, B 0.000, C 0.000 }
gfCNCPoint6[11226] = {X 403.0811, Y 13.9219, Z -8.0000, A 0.000, B 0.000, C 0.000 }
gfCNCPoint6[11227] = {X 402.7551, Y 14.8144, Z -8.0000, A 0.000, B 0.000, C 0.000 }
gfCNCPoint6[11228] = {X 405.3487, Y 19.2892, Z -8.0000, A 0.000, B 0.000, C 0.000 }
gfCNCPoint6[11229] = {X 408.1455, Y 14.7688, Z -8.0000, A 0.000, B 0.000, C 0.000 }
gfCNCPoint6[11230] = {X 408.1087, Y 14.6914, Z -8.0000, A 0.000, B 0.000, C 0.000 }
gfCNCPoint6[11231] = {X 408.0736, Y 14.6132, Z -8.0000, A 0.000, B 0.000, C 0.000 }
gfCNCPoint6[11232] = {X 407.8216, Y 13.8305, Z -8.0000, A 0.000, B 0.000, C 0.000 }
gfCNCPoint6[11233] = {X 407.7317, Y 13.0131, Z -8.0000, A 0.000, B 0.000, C 0.000 }
gfCNCPoint6[11234] = {X 407.7315, Y 12.1868, Z -8.0000, A 0.000, B 0.000, C 0.000 }
gfCNCPoint6[11235] = {X 407.8338, Y 11.2789, Z -8.0000, A 0.000, B 0.000, C 0.000 }
gfCNCPoint6[11236] = {X 408.1356, Y 10.4166, Z -8.0000, A 0.000, B 0.000, C 0.000 }
gfCNCPoint6[11237] = {X 408.6217, Y 9.6430, Z -8.0000, A 0.000, B 0.000, C 0.000 }
gfCNCPoint6[11238] = {X 409.2677, Y 8.9969, Z -8.0000, A 0.000, B 0.000, C 0.000 }
gfCNCPoint6[11239] = {X 410.0413, Y 8.5109, Z -8.0000, A 0.000, B 0.000, C 0.000 }
gfCNCPoint6[11240] = {X 410.9037, Y 8.2091, Z -8.0000, A 0.000, B 0.000, C 0.000 }
gfCNCPoint6[11241] = {X 411.8115, Y 8.1068, Z -8.0000, A 0.000, B 0.000, C 0.000 }
gfCNCPoint6[11242] = {X 419.3245, Y 8.1068, Z -8.0000, A 0.000, B 0.000, C 0.000 }
gfCNCPoint6[11243] = {X 420.2323, Y 8.2091, Z -8.0000, A 0.000, B 0.000, C 0.000 }
gfCNCPoint6[11244] = {X 421.0947, Y 8.5109, Z -8.0000, A 0.000, B 0.000, C 0.000 }
gfCNCPoint6[11245] = {X 421.8683, Y 8.9969, Z -8.0000, A 0.000, B 0.000, C 0.000 }
gfCNCPoint6[11246] = {X 422.5143, Y 9.6430, Z -8.0000, A 0.000, B 0.000, C 0.000 }
gfCNCPoint6[11247] = {X 423.0004, Y 10.4166, Z -8.0000, A 0.000, B 0.000, C 0.000 }
gfCNCPoint6[11248] = {X 423.3022, Y 11.2789, Z -8.0000, A 0.000, B 0.000, C 0.000 }
gfCNCPoint6[11249] = {X 423.4045, Y 12.1868, Z -8.0000, A 0.000, B 0.000, C 0.000 }
gfCNCPoint6[11250] = {X 423.4045, Y 12.9785, Z -8.0000, A 0.000, B 0.000, C 0.000 }
gfCNCPoint6[11251] = {X 423.3150, Y 13.8081, Z -8.0000, A 0.000, B 0.000, C 0.000 }
gfCNCPoint6[11252] = {X 423.0611, Y 14.6028, Z -8.0000, A 0.000, B 0.000, C 0.000 }
gfCNCPoint6[11253] = {X 422.6529, Y 15.3305, Z -8.0000, A 0.000, B 0.000, C 0.000 }
gfCNCPoint6[11254] = {X 422.1071, Y 15.9616, Z -8.0000, A 0.000, B 0.000, C 0.000 }
gfCNCPoint6[11255] = {X 421.4458, Y 16.4704, Z -8.0000, A 0.000, B 0.000, C 0.000 }
gfCNCPoint6[11256] = {X 420.6960, Y 16.8363, Z -8.0000, A 0.000, B 0.000, C 0.000 }
gfCNCPoint6[11257] = {X 419.9477, Y 17.8364, Z -8.0000, A 0.000, B 0.000, C 0.000 }
gfCNCPoint6[11258] = {X 419.2723, Y 18.8871, Z -8.0000, A 0.000, B 0.000, C 0.000 }
gfCNCPoint6[11259] = {X 417.7903, Y 21.2859, Z -8.0000, A 0.000, B 0.000, C 0.000 }
gfCNCPoint6[11260] = {X 415.9479, Y 24.2449, Z -8.0000, A 0.000, B 0.000, C 0.000 }
gfCNCPoint6[11261] = {X 419.3436, Y 26.3590, Z -8.0000, A 0.000, B 0.000, C 0.000 }
gfCNCPoint6[11262] = {X 415.8800, Y 24.2026, Z -8.0000, A 0.000, B 0.000, C 0.000 }
gfCNCPoint6[11263] = {X 411.2282, Y 31.6740, Z -8.0000, A 0.000, B 0.000, C 0.000 }
gfCNCPoint6[11264] = {X 411.2288, Y 41.0466, Z -8.0000, A 0.000, B 0.000, C 0.000 }
gfCNCPoint6[11265] = {X 411.8653, Y 41.6900, Z -8.0000, A 0.000, B 0.000, C 0.000 }
gfCNCPoint6[11266] = {X 412.3458, Y 42.4569, Z -8.0000, A 0.000, B 0.000, C 0.000 }
gfCNCPoint6[11267] = {X 412.6471, Y 43.3102, Z -8.0000, A 0.000, B 0.000, C 0.000 }
gfCNCPoint6[11268] = {X 412.7547, Y 44.2088, Z -8.0000, A 0.000, B 0.000, C 0.000 }
gfCNCPoint6[11269] = {X 412.7545, Y 45.0384, Z -8.0000, A 0.000, B 0.000, C 0.000 }
gfCNCPoint6[11270] = {X 412.6469, Y 45.9222, Z -8.0000, A 0.000, B 0.000, C 0.000 }
gfCNCPoint6[11271] = {X 412.3466, Y 46.7602, Z -8.0000, A 0.000, B 0.000, C 0.000 }
gfCNCPoint6[11272] = {X 411.8683, Y 47.5111, Z -8.0000, A 0.000, B 0.000, C 0.000 }
gfCNCPoint6[11273] = {X 411.2357, Y 48.1376, Z -8.0000, A 0.000, B 0.000, C 0.000 }
gfCNCPoint6[11274] = {X 410.4803, Y 48.6086, Z -8.0000, A 0.000, B 0.000, C 0.000 }
gfCNCPoint6[11275] = {X 409.6394, Y 48.9009, Z -8.0000, A 0.000, B 0.000, C 0.000 }
gfCNCPoint6[11276] = {X 408.7547, Y 49.0000, Z -8.0000, A 0.000, B 0.000, C 0.000 }
gfCNCPoint6[11277] = {X 402.3112, Y 49.0000, Z -8.0000, A 0.000, B 0.000, C 0.000 }
gfCNCPoint6[11278] = {X 401.4211, Y 48.8997, Z -8.0000, A 0.000, B 0.000, C 0.000 }
gfCNCPoint6[11279] = {X 400.5757, Y 48.6039, Z -8.0000, A 0.000, B 0.000, C 0.000 }
gfCNCPoint6[11280] = {X 399.8172, Y 48.1273, Z -8.0000, A 0.000, B 0.000, C 0.000 }
gfCNCPoint6[11281] = {X 399.1839, Y 47.4939, Z -8.0000, A 0.000, B 0.000, C 0.000 }
gfCNCPoint6[11282] = {X 398.7073, Y 46.7355, Z -8.0000, A 0.000, B 0.000, C 0.000 }
gfCNCPoint6[11283] = {X 398.4115, Y 45.8901, Z -8.0000, A 0.000, B 0.000, C 0.000 }
gfCNCPoint6[11284] = {X 398.3112, Y 45.0000, Z -8.0000, A 0.000, B 0.000, C 0.000 }
gfCNCPoint6[11285] = {X 398.3115, Y 44.1569, Z -8.0000, A 0.000, B 0.000, C 0.000 }
gfCNCPoint6[11286] = {X 398.4217, Y 43.2753, Z -8.0000, A 0.000, B 0.000, C 0.000 }
gfCNCPoint6[11287] = {X 398.7237, Y 42.4397, Z -8.0000, A 0.000, B 0.000, C 0.000 }
gfCNCPoint6[11288] = {X 399.2028, Y 41.6913, Z -8.0000, A 0.000, B 0.000, C 0.000 }
gfCNCPoint6[11289] = {X 399.8352, Y 41.0672, Z -8.0000, A 0.000, B 0.000, C 0.000 }
gfCNCPoint6[11290] = {X 399.8360, Y 31.5925, Z -8.0000, A 0.000, B 0.000, C 0.000 }
gfCNCPoint6[11291] = {X 393.7120, Y 20.9428, Z -8.0000, A 0.000, B 0.000, C 0.000 }
gfCNCPoint6[11292] = {X 392.8604, Y 19.4956, Z -8.0000, A 0.000, B 0.000, C 0.000 }
gfCNCPoint6[11293] = {X 391.9801, Y 18.0658, Z -8.0000, A 0.000, B 0.000, C 0.000 }
gfCNCPoint6[11294] = {X 391.4559, Y 17.3417, Z -8.0000, A 0.000, B 0.000, C 0.000 }
gfCNCPoint6[11295] = {X 390.8426, Y 16.6913, Z -8.0000, A 0.000, B 0.000, C 0.000 }
gfCNCPoint6[11296] = {X 390.0091, Y 16.2361, Z -8.0000, A 0.000, B 0.000, C 0.000 }
gfCNCPoint6[11297] = {X 389.3064, Y 15.5972, Z -8.0000, A 0.000, B 0.000, C 0.000 }
gfCNCPoint6[11298] = {X 388.7742, Y 14.8107, Z -8.0000, A 0.000, B 0.000, C 0.000 }
gfCNCPoint6[11299] = {X 388.4424, Y 13.9209, Z -8.0000, A 0.000, B 0.000, C 0.000 }
gfCNCPoint6[11300] = {X 388.3296, Y 12.9780, Z -8.0000, A 0.000, B 0.000, C 0.000 }
gfCNCPoint6[11301] = {X 388.3296, Y 12.1868, Z -8.0000, A 0.000, B 0.000, C 0.000 }
gfCNCPoint6[11302] = {X 388.4299, Y 11.2967, Z -8.0000, A 0.000, B 0.000, C 0.000 }
gfCNCPoint6[11303] = {X 388.7258, Y 10.4513, Z -8.0000, A 0.000, B 0.000, C 0.000 }
gfCNCPoint6[11304] = {X 389.2023, Y 9.6929, Z -8.0000, A 0.000, B 0.000, C 0.000 }
gfCNCPoint6[11305] = {X 389.8357, Y 9.0595, Z -8.0000, A 0.000, B 0.000, C 0.000 }
gfCNCPoint6[11306] = {X 390.5941, Y 8.5829, Z -8.0000, A 0.000, B 0.000, C 0.000 }
gfCNCPoint6[11307] = {X 391.4395, Y 8.2871, Z -8.0000, A 0.000, B 0.000, C 0.000 }
gfCNCPoint6[11308] = {X 392.3296, Y 8.1868, Z -8.0000, A 0.000, B 0.000, C 0.000 }
gfCNCPoint6[11309] = {X 399.1118, Y 8.1868, Z -8.0000, A 0.000, B 0.000, C 0.000 }
gfCNCPoint6[11310] = {X 400.0018, Y 8.2871, Z -8.0000, A 0.000, B 0.000, C 0.000 }
gfCNCPoint6[11311] = {X 400.8473, Y 8.5829, Z -8.0000, A 0.000, B 0.000, C 0.000 }
gfCNCPoint6[11312] = {X 401.6057, Y 9.0595, Z -8.0000, A 0.000, B 0.000, C 0.000 }
gfCNCPoint6[11313] = {X 402.2391, Y 9.6929, Z -8.0000, A 0.000, B 0.000, C 0.000 }
gfCNCPoint6[11314] = {X 402.7156, Y 10.4513, Z -8.0000, A 0.000, B 0.000, C 0.000 }
gfCNCPoint6[11315] = {X 403.0115, Y 11.2967, Z -8.0000, A 0.000, B 0.000, C 0.000 }
gfCNCPoint6[11316] = {X 403.1118, Y 12.1868, Z -8.0000, A 0.000, B 0.000, C 0.000 }
gfCNCPoint6[11317] = {X 403.1115, Y 13.0192, Z -8.0000, A 0.000, B 0.000, C 0.000 }
gfCNCPoint6[11318] = {X 402.9933, Y 13.9442, Z -8.0000, A 0.000, B 0.000, C 0.000 }
gfCNCPoint6[11319] = {X 402.6641, Y 14.8167, Z -8.0000, A 0.000, B 0.000, C 0.000 }
gfCNCPoint6[11320] = {X 405.2576, Y 19.3199, Z -8.0000, A 0.000, B 0.000, C 0.000 }
gfCNCPoint6[11321] = {X 405.3700, Y 19.4069, Z -8.0000, A 0.000, B 0.000, C 0.000 }
gfCNCPoint6[11322] = {X 408.1933, Y 14.8341, Z -8.0000, A 0.000, B 0.000, C 0.000 }
gfCNCPoint6[11323] = {X 408.2428, Y 14.7847, Z -8.0000, A 0.000, B 0.000, C 0.000 }
gfCNCPoint6[11324] = {X 408.1934, Y 14.6836, Z -8.0000, A 0.000, B 0.000, C 0.000 }
gfCNCPoint6[11325] = {X 408.1469, Y 14.5812, Z -8.0000, A 0.000, B 0.000, C 0.000 }
gfCNCPoint6[11326] = {X 407.8963, Y 13.7969, Z -8.0000, A 0.000, B 0.000, C 0.000 }
gfCNCPoint6[11327] = {X 407.8115, Y 12.9780, Z -8.0000, A 0.000, B 0.000, C 0.000 }
gfCNCPoint6[11328] = {X 407.8115, Y 12.1868, Z -8.0000, A 0.000, B 0.000, C 0.000 }
gfCNCPoint6[11329] = {X 407.9118, Y 11.2967, Z -8.0000, A 0.000, B 0.000, C 0.000 }
gfCNCPoint6[11330] = {X 408.2077, Y 10.4513, Z -8.0000, A 0.000, B 0.000, C 0.000 }
gfCNCPoint6[11331] = {X 408.6842, Y 9.6929, Z -8.0000, A 0.000, B 0.000, C 0.000 }
gfCNCPoint6[11332] = {X 409.3176, Y 9.0595, Z -8.0000, A 0.000, B 0.000, C 0.000 }
gfCNCPoint6[11333] = {X 410.0760, Y 8.5829, Z -8.0000, A 0.000, B 0.000, C 0.000 }
gfCNCPoint6[11334] = {X 410.9215, Y 8.2871, Z -8.0000, A 0.000, B 0.000, C 0.000 }
gfCNCPoint6[11335] = {X 411.8115, Y 8.1868, Z -8.0000, A 0.000, B 0.000, C 0.000 }
gfCNCPoint6[11336] = {X 419.3245, Y 8.1868, Z -8.0000, A 0.000, B 0.000, C 0.000 }
gfCNCPoint6[11337] = {X 420.2145, Y 8.2871, Z -8.0000, A 0.000, B 0.000, C 0.000 }
gfCNCPoint6[11338] = {X 421.0600, Y 8.5829, Z -8.0000, A 0.000, B 0.000, C 0.000 }
gfCNCPoint6[11339] = {X 421.8184, Y 9.0595, Z -8.0000, A 0.000, B 0.000, C 0.000 }
gfCNCPoint6[11340] = {X 422.4518, Y 9.6929, Z -8.0000, A 0.000, B 0.000, C 0.000 }
gfCNCPoint6[11341] = {X 422.9283, Y 10.4513, Z -8.0000, A 0.000, B 0.000, C 0.000 }
gfCNCPoint6[11342] = {X 423.2242, Y 11.2967, Z -8.0000, A 0.000, B 0.000, C 0.000 }
gfCNCPoint6[11343] = {X 423.3245, Y 12.1868, Z -8.0000, A 0.000, B 0.000, C 0.000 }
gfCNCPoint6[11344] = {X 423.3245, Y 12.9780, Z -8.0000, A 0.000, B 0.000, C 0.000 }
gfCNCPoint6[11345] = {X 423.2360, Y 13.7951, Z -8.0000, A 0.000, B 0.000, C 0.000 }
gfCNCPoint6[11346] = {X 422.9848, Y 14.5777, Z -8.0000, A 0.000, B 0.000, C 0.000 }
gfCNCPoint6[11347] = {X 422.5811, Y 15.2936, Z -8.0000, A 0.000, B 0.000, C 0.000 }
gfCNCPoint6[11348] = {X 422.0415, Y 15.9135, Z -8.0000, A 0.000, B 0.000, C 0.000 }
gfCNCPoint6[11349] = {X 421.3881, Y 16.4120, Z -8.0000, A 0.000, B 0.000, C 0.000 }
gfCNCPoint6[11350] = {X 420.6477, Y 16.7687, Z -8.0000, A 0.000, B 0.000, C 0.000 }
gfCNCPoint6[11351] = {X 419.8885, Y 17.7813, Z -8.0000, A 0.000, B 0.000, C 0.000 }
gfCNCPoint6[11352] = {X 419.2039, Y 18.8457, Z -8.0000, A 0.000, B 0.000, C 0.000 }
gfCNCPoint6[11353] = {X 417.7223, Y 21.2437, Z -8.0000, A 0.000, B 0.000, C 0.000 }
gfCNCPoint6[11354] = {X 415.8800, Y 24.2026, Z -8.0000, A 0.000, B 0.000, C 0.000 }
gfCNCPoint6[11355] = {X 419.3436, Y 26.3590, Z -8.0000, A 0.000, B 0.000, C 0.000 }
gfCNCPoint6[11356] = {X 419.3436, Y 26.3590, Z -5.0000, A 0.000, B 0.000, C 0.000 }
gfCNCPoint6[11357] = {X 419.3436, Y 26.3590, Z 11.0000, A 0.000, B 0.000, C 0.000 }
gfCNCPoint6[11358] = {X 368.0085, Y 43.6796, Z 11.0000, A 0.000, B 0.000, C 0.000 }
gfCNCPoint6[11359] = {X 368.0085, Y 43.6796, Z -5.0000, A 0.000, B 0.000, C 0.000 }
gfCNCPoint6[11360] = {X 368.0085, Y 43.6796, Z -8.0000, A 0.000, B 0.000, C 0.000 }
gfCNCPoint6[11361] = {X 364.7162, Y 41.2699, Z -8.0000, A 0.000, B 0.000, C 0.000 }
gfCNCPoint6[11362] = {X 364.6579, Y 41.3495, Z -8.0000, A 0.000, B 0.000, C 0.000 }
gfCNCPoint6[11363] = {X 363.2575, Y 43.0264, Z -8.0000, A 0.000, B 0.000, C 0.000 }
gfCNCPoint6[11364] = {X 361.6976, Y 44.5561, Z -8.0000, A 0.000, B 0.000, C 0.000 }
gfCNCPoint6[11365] = {X 359.9935, Y 45.9234, Z -8.0000, A 0.000, B 0.000, C 0.000 }
gfCNCPoint6[11366] = {X 358.1622, Y 47.1148, Z -8.0000, A 0.000, B 0.000, C 0.000 }
gfCNCPoint6[11367] = {X 356.2216, Y 48.1185, Z -8.0000, A 0.000, B 0.000, C 0.000 }
gfCNCPoint6[11368] = {X 354.0239, Y 48.9388, Z -8.0000, A 0.000, B 0.000, C 0.000 }
gfCNCPoint6[11369] = {X 351.7542, Y 49.5312, Z -8.0000, A 0.000, B 0.000, C 0.000 }
gfCNCPoint6[11370] = {X 349.4359, Y 49.8896, Z -8.0000, A 0.000, B 0.000, C 0.000 }
gfCNCPoint6[11371] = {X 347.0933, Y 50.0103, Z -8.0000, A 0.000, B 0.000, C 0.000 }
gfCNCPoint6[11372] = {X 345.0267, Y 49.9754, Z -8.0000, A 0.000, B 0.000, C 0.000 }
gfCNCPoint6[11373] = {X 342.9709, Y 49.7614, Z -8.0000, A 0.000, B 0.000, C 0.000 }
gfCNCPoint6[11374] = {X 340.9414, Y 49.3699, Z -8.0000, A 0.000, B 0.000, C 0.000 }
gfCNCPoint6[11375] = {X 338.9535, Y 48.8039, Z -8.0000, A 0.000, B 0.000, C 0.000 }
gfCNCPoint6[11376] = {X 337.0222, Y 48.0677, Z -8.0000, A 0.000, B 0.000, C 0.000 }
gfCNCPoint6[11377] = {X 335.1621, Y 47.1667, Z -8.0000, A 0.000, B 0.000, C 0.000 }
gfCNCPoint6[11378] = {X 333.5779, Y 46.1885, Z -8.0000, A 0.000, B 0.000, C 0.000 }
gfCNCPoint6[11379] = {X 332.0750, Y 45.0897, Z -8.0000, A 0.000, B 0.000, C 0.000 }
gfCNCPoint6[11380] = {X 330.6624, Y 43.8770, Z -8.0000, A 0.000, B 0.000, C 0.000 }
gfCNCPoint6[11381] = {X 329.7213, Y 43.8764, Z -8.0000, A 0.000, B 0.000, C 0.000 }
gfCNCPoint6[11382] = {X 328.8027, Y 43.6721, Z -8.0000, A 0.000, B 0.000, C 0.000 }
gfCNCPoint6[11383] = {X 327.9501, Y 43.2738, Z -8.0000, A 0.000, B 0.000, C 0.000 }
gfCNCPoint6[11384] = {X 327.2040, Y 42.7002, Z -8.0000, A 0.000, B 0.000, C 0.000 }
gfCNCPoint6[11385] = {X 326.5808, Y 42.0925, Z -8.0000, A 0.000, B 0.000, C 0.000 }
gfCNCPoint6[11386] = {X 325.9523, Y 41.3190, Z -8.0000, A 0.000, B 0.000, C 0.000 }
gfCNCPoint6[11387] = {X 325.5179, Y 40.4220, Z -8.0000, A 0.000, B 0.000, C 0.000 }
gfCNCPoint6[11388] = {X 325.3006, Y 39.4493, Z -8.0000, A 0.000, B 0.000, C 0.000 }
gfCNCPoint6[11389] = {X 325.3120, Y 38.4527, Z -8.0000, A 0.000, B 0.000, C 0.000 }
gfCNCPoint6[11390] = {X 325.5514, Y 37.4852, Z -8.0000, A 0.000, B 0.000, C 0.000 }
gfCNCPoint6[11391] = {X 326.0062, Y 36.5984, Z -8.0000, A 0.000, B 0.000, C 0.000 }
gfCNCPoint6[11392] = {X 330.2396, Y 30.2686, Z -8.0000, A 0.000, B 0.000, C 0.000 }
gfCNCPoint6[11393] = {X 330.8410, Y 29.5518, Z -8.0000, A 0.000, B 0.000, C 0.000 }
gfCNCPoint6[11394] = {X 331.5826, Y 28.9812, Z -8.0000, A 0.000, B 0.000, C 0.000 }
gfCNCPoint6[11395] = {X 332.4297, Y 28.5837, Z -8.0000, A 0.000, B 0.000, C 0.000 }
gfCNCPoint6[11396] = {X 333.3425, Y 28.3780, Z -8.0000, A 0.000, B 0.000, C 0.000 }
gfCNCPoint6[11397] = {X 334.2782, Y 28.3736, Z -8.0000, A 0.000, B 0.000, C 0.000 }
gfCNCPoint6[11398] = {X 335.1929, Y 28.5708, Z -8.0000, A 0.000, B 0.000, C 0.000 }
gfCNCPoint6[11399] = {X 336.0437, Y 28.9604, Z -8.0000, A 0.000, B 0.000, C 0.000 }
gfCNCPoint6[11400] = {X 336.7907, Y 29.5240, Z -8.0000, A 0.000, B 0.000, C 0.000 }
gfCNCPoint6[11401] = {X 337.4284, Y 30.1382, Z -8.0000, A 0.000, B 0.000, C 0.000 }
gfCNCPoint6[11402] = {X 338.0536, Y 30.9133, Z -8.0000, A 0.000, B 0.000, C 0.000 }
gfCNCPoint6[11403] = {X 338.4846, Y 31.8110, Z -8.0000, A 0.000, B 0.000, C 0.000 }
gfCNCPoint6[11404] = {X 338.6987, Y 32.7835, Z -8.0000, A 0.000, B 0.000, C 0.000 }
gfCNCPoint6[11405] = {X 338.6844, Y 33.7792, Z -8.0000, A 0.000, B 0.000, C 0.000 }
gfCNCPoint6[11406] = {X 338.7027, Y 33.8726, Z -8.0000, A 0.000, B 0.000, C 0.000 }
gfCNCPoint6[11407] = {X 339.4938, Y 34.5959, Z -8.0000, A 0.000, B 0.000, C 0.000 }
gfCNCPoint6[11408] = {X 340.6305, Y 35.5019, Z -8.0000, A 0.000, B 0.000, C 0.000 }
gfCNCPoint6[11409] = {X 341.8796, Y 36.2452, Z -8.0000, A 0.000, B 0.000, C 0.000 }
gfCNCPoint6[11410] = {X 343.2181, Y 36.8121, Z -8.0000, A 0.000, B 0.000, C 0.000 }
gfCNCPoint6[11411] = {X 344.6211, Y 37.1922, Z -8.0000, A 0.000, B 0.000, C 0.000 }
gfCNCPoint6[11412] = {X 346.0627, Y 37.3782, Z -8.0000, A 0.000, B 0.000, C 0.000 }
gfCNCPoint6[11413] = {X 347.5162, Y 37.3669, Z -8.0000, A 0.000, B 0.000, C 0.000 }
gfCNCPoint6[11414] = {X 348.9573, Y 37.1738, Z -8.0000, A 0.000, B 0.000, C 0.000 }
gfCNCPoint6[11415] = {X 350.3476, Y 36.7484, Z -8.0000, A 0.000, B 0.000, C 0.000 }
gfCNCPoint6[11416] = {X 351.6501, Y 36.1022, Z -8.0000, A 0.000, B 0.000, C 0.000 }
gfCNCPoint6[11417] = {X 352.8298, Y 35.2525, Z -8.0000, A 0.000, B 0.000, C 0.000 }
gfCNCPoint6[11418] = {X 353.9828, Y 34.1319, Z -8.0000, A 0.000, B 0.000, C 0.000 }
gfCNCPoint6[11419] = {X 354.9806, Y 32.8712, Z -8.0000, A 0.000, B 0.000, C 0.000 }
gfCNCPoint6[11420] = {X 355.8063, Y 31.4917, Z -8.0000, A 0.000, B 0.000, C 0.000 }
gfCNCPoint6[11421] = {X 356.4460, Y 30.0166, Z -8.0000, A 0.000, B 0.000, C 0.000 }
gfCNCPoint6[11422] = {X 356.8888, Y 28.4710, Z -8.0000, A 0.000, B 0.000, C 0.000 }
gfCNCPoint6[11423] = {X 357.1621, Y 26.7828, Z -8.0000, A 0.000, B 0.000, C 0.000 }
gfCNCPoint6[11424] = {X 357.2734, Y 25.0763, Z -8.0000, A 0.000, B 0.000, C 0.000 }
gfCNCPoint6[11425] = {X 357.2217, Y 23.3668, Z -8.0000, A 0.000, B 0.000, C 0.000 }
gfCNCPoint6[11426] = {X 357.0075, Y 21.6701, Z -8.0000, A 0.000, B 0.000, C 0.000 }
gfCNCPoint6[11427] = {X 356.6539, Y 20.1544, Z -8.0000, A 0.000, B 0.000, C 0.000 }
gfCNCPoint6[11428] = {X 356.1045, Y 18.6982, Z -8.0000, A 0.000, B 0.000, C 0.000 }
gfCNCPoint6[11429] = {X 355.3687, Y 17.3267, Z -8.0000, A 0.000, B 0.000, C 0.000 }
gfCNCPoint6[11430] = {X 354.4594, Y 16.0636, Z -8.0000, A 0.000, B 0.000, C 0.000 }
gfCNCPoint6[11431] = {X 353.5888, Y 15.1366, Z -8.0000, A 0.000, B 0.000, C 0.000 }
gfCNCPoint6[11432] = {X 352.5980, Y 14.3394, Z -8.0000, A 0.000, B 0.000, C 0.000 }
gfCNCPoint6[11433] = {X 351.5062, Y 13.6872, Z -8.0000, A 0.000, B 0.000, C 0.000 }
gfCNCPoint6[11434] = {X 350.3346, Y 13.1926, Z -8.0000, A 0.000, B 0.000, C 0.000 }
gfCNCPoint6[11435] = {X 349.1057, Y 12.8654, Z -8.0000, A 0.000, B 0.000, C 0.000 }
gfCNCPoint6[11436] = {X 347.3453, Y 12.6454, Z -8.0000, A 0.000, B 0.000, C 0.000 }
gfCNCPoint6[11437] = {X 345.5712, Y 12.6607, Z -8.0000, A 0.000, B 0.000, C 0.000 }
gfCNCPoint6[11438] = {X 343.8148, Y 12.9108, Z -8.0000, A 0.000, B 0.000, C 0.000 }
gfCNCPoint6[11439] = {X 342.1070, Y 13.3915, Z -8.0000, A 0.000, B 0.000, C 0.000 }
gfCNCPoint6[11440] = {X 340.4779, Y 14.0942, Z -8.0000, A 0.000, B 0.000, C 0.000 }
gfCNCPoint6[11441] = {X 338.9564, Y 15.0065, Z -8.0000, A 0.000, B 0.000, C 0.000 }
gfCNCPoint6[11442] = {X 338.9173, Y 15.8510, Z -8.0000, A 0.000, B 0.000, C 0.000 }
gfCNCPoint6[11443] = {X 338.7146, Y 16.6716, Z -8.0000, A 0.000, B 0.000, C 0.000 }
gfCNCPoint6[11444] = {X 338.3559, Y 17.4371, Z -8.0000, A 0.000, B 0.000, C 0.000 }
gfCNCPoint6[11445] = {X 337.8551, Y 18.1180, Z -8.0000, A 0.000, B 0.000, C 0.000 }
gfCNCPoint6[11446] = {X 337.2312, Y 18.6884, Z -8.0000, A 0.000, B 0.000, C 0.000 }
gfCNCPoint6[11447] = {X 336.5140, Y 19.2162, Z -8.0000, A 0.000, B 0.000, C 0.000 }
gfCNCPoint6[11448] = {X 335.6982, Y 19.6754, Z -8.0000, A 0.000, B 0.000, C 0.000 }
gfCNCPoint6[11449] = {X 334.8027, Y 19.9480, Z -8.0000, A 0.000, B 0.000, C 0.000 }
gfCNCPoint6[11450] = {X 333.8694, Y 20.0213, Z -8.0000, A 0.000, B 0.000, C 0.000 }
gfCNCPoint6[11451] = {X 332.9422, Y 19.8919, Z -8.0000, A 0.000, B 0.000, C 0.000 }
gfCNCPoint6[11452] = {X 332.0647, Y 19.5657, Z -8.0000, A 0.000, B 0.000, C 0.000 }
gfCNCPoint6[11453] = {X 331.2781, Y 19.0581, Z -8.0000, A 0.000, B 0.000, C 0.000 }
gfCNCPoint6[11454] = {X 330.6193, Y 18.3931, Z -8.0000, A 0.000, B 0.000, C 0.000 }
gfCNCPoint6[11455] = {X 330.1192, Y 17.6017, Z -8.0000, A 0.000, B 0.000, C 0.000 }
gfCNCPoint6[11456] = {X 326.5942, Y 10.3502, Z -8.0000, A 0.000, B 0.000, C 0.000 }
gfCNCPoint6[11457] = {X 326.2930, Y 9.5271, Z -8.0000, A 0.000, B 0.000, C 0.000 }
gfCNCPoint6[11458] = {X 326.1640, Y 8.6602, Z -8.0000, A 0.000, B 0.000, C 0.000 }
gfCNCPoint6[11459] = {X 326.2128, Y 7.7851, Z -8.0000, A 0.000, B 0.000, C 0.000 }
gfCNCPoint6[11460] = {X 326.4371, Y 6.9378, Z -8.0000, A 0.000, B 0.000, C 0.000 }
gfCNCPoint6[11461] = {X 326.8279, Y 6.1532, Z -8.0000, A 0.000, B 0.000, C 0.000 }
gfCNCPoint6[11462] = {X 327.3690, Y 5.4637, Z -8.0000, A 0.000, B 0.000, C 0.000 }
gfCNCPoint6[11463] = {X 328.0381, Y 4.8976, Z -8.0000, A 0.000, B 0.000, C 0.000 }
gfCNCPoint6[11464] = {X 328.7084, Y 4.4386, Z -8.0000, A 0.000, B 0.000, C 0.000 }
gfCNCPoint6[11465] = {X 329.5886, Y 3.9823, Z -8.0000, A 0.000, B 0.000, C 0.000 }
gfCNCPoint6[11466] = {X 330.5496, Y 3.7388, Z -8.0000, A 0.000, B 0.000, C 0.000 }
gfCNCPoint6[11467] = {X 331.5409, Y 3.7207, Z -8.0000, A 0.000, B 0.000, C 0.000 }
gfCNCPoint6[11468] = {X 332.5101, Y 3.9291, Z -8.0000, A 0.000, B 0.000, C 0.000 }
gfCNCPoint6[11469] = {X 333.9835, Y 3.1055, Z -8.0000, A 0.000, B 0.000, C 0.000 }
gfCNCPoint6[11470] = {X 335.5040, Y 2.3725, Z -8.0000, A 0.000, B 0.000, C 0.000 }
gfCNCPoint6[11471] = {X 337.6430, Y 1.5021, Z -8.0000, A 0.000, B 0.000, C 0.000 }
gfCNCPoint6[11472] = {X 339.8502, Y 0.8229, Z -8.0000, A 0.000, B 0.000, C 0.000 }
gfCNCPoint6[11473] = {X 342.1086, Y 0.3401, Z -8.0000, A 0.000, B 0.000, C 0.000 }
gfCNCPoint6[11474] = {X 344.4005, Y 0.0573, Z -8.0000, A 0.000, B 0.000, C 0.000 }
gfCNCPoint6[11475] = {X 346.7085, Y -0.0231, Z -8.0000, A 0.000, B 0.000, C 0.000 }
gfCNCPoint6[11476] = {X 349.0146, Y 0.0994, Z -8.0000, A 0.000, B 0.000, C 0.000 }
gfCNCPoint6[11477] = {X 351.3010, Y 0.4239, Z -8.0000, A 0.000, B 0.000, C 0.000 }
gfCNCPoint6[11478] = {X 353.2151, Y 0.8471, Z -8.0000, A 0.000, B 0.000, C 0.000 }
gfCNCPoint6[11479] = {X 355.0815, Y 1.4468, Z -8.0000, A 0.000, B 0.000, C 0.000 }
gfCNCPoint6[11480] = {X 356.8839, Y 2.2178, Z -8.0000, A 0.000, B 0.000, C 0.000 }
gfCNCPoint6[11481] = {X 358.6066, Y 3.1533, Z -8.0000, A 0.000, B 0.000, C 0.000 }
gfCNCPoint6[11482] = {X 360.2347, Y 4.2452, Z -8.0000, A 0.000, B 0.000, C 0.000 }
gfCNCPoint6[11483] = {X 361.7540, Y 5.4840, Z -8.0000, A 0.000, B 0.000, C 0.000 }
gfCNCPoint6[11484] = {X 363.1514, Y 6.8589, Z -8.0000, A 0.000, B 0.000, C 0.000 }
gfCNCPoint6[11485] = {X 364.6986, Y 8.7281, Z -8.0000, A 0.000, B 0.000, C 0.000 }
gfCNCPoint6[11486] = {X 366.0557, Y 10.7397, Z -8.0000, A 0.000, B 0.000, C 0.000 }
gfCNCPoint6[11487] = {X 367.2096, Y 12.8743, Z -8.0000, A 0.000, B 0.000, C 0.000 }
gfCNCPoint6[11488] = {X 368.1494, Y 15.1114, Z -8.0000, A 0.000, B 0.000, C 0.000 }
gfCNCPoint6[11489] = {X 368.8659, Y 17.4297, Z -8.0000, A 0.000, B 0.000, C 0.000 }
gfCNCPoint6[11490] = {X 369.3482, Y 19.7225, Z -8.0000, A 0.000, B 0.000, C 0.000 }
gfCNCPoint6[11491] = {X 369.6592, Y 22.0446, Z -8.0000, A 0.000, B 0.000, C 0.000 }
gfCNCPoint6[11492] = {X 369.7972, Y 24.3835, Z -8.0000, A 0.000, B 0.000, C 0.000 }
gfCNCPoint6[11493] = {X 369.7614, Y 26.7261, Z -8.0000, A 0.000, B 0.000, C 0.000 }
gfCNCPoint6[11494] = {X 369.5521, Y 29.0596, Z -8.0000, A 0.000, B 0.000, C 0.000 }
gfCNCPoint6[11495] = {X 369.1703, Y 31.3712, Z -8.0000, A 0.000, B 0.000, C 0.000 }
gfCNCPoint6[11496] = {X 368.6462, Y 33.4755, Z -8.0000, A 0.000, B 0.000, C 0.000 }
gfCNCPoint6[11497] = {X 367.9383, Y 35.5252, Z -8.0000, A 0.000, B 0.000, C 0.000 }
gfCNCPoint6[11498] = {X 367.0522, Y 37.5044, Z -8.0000, A 0.000, B 0.000, C 0.000 }
gfCNCPoint6[11499] = {X 365.9948, Y 39.3977, Z -8.0000, A 0.000, B 0.000, C 0.000 }
gfCNCPoint6[11500] = {X 364.7744, Y 41.1902, Z -8.0000, A 0.000, B 0.000, C 0.000 }
gfCNCPoint6[11501] = {X 364.7162, Y 41.2699, Z -8.0000, A 0.000, B 0.000, C 0.000 }
gfCNCPoint6[11502] = {X 367.9439, Y 43.6324, Z -8.0000, A 0.000, B 0.000, C 0.000 }
gfCNCPoint6[11503] = {X 364.6516, Y 41.2226, Z -8.0000, A 0.000, B 0.000, C 0.000 }
gfCNCPoint6[11504] = {X 364.5937, Y 41.3018, Z -8.0000, A 0.000, B 0.000, C 0.000 }
gfCNCPoint6[11505] = {X 363.1985, Y 42.9724, Z -8.0000, A 0.000, B 0.000, C 0.000 }
gfCNCPoint6[11506] = {X 361.6444, Y 44.4963, Z -8.0000, A 0.000, B 0.000, C 0.000 }
gfCNCPoint6[11507] = {X 359.9468, Y 45.8584, Z -8.0000, A 0.000, B 0.000, C 0.000 }
gfCNCPoint6[11508] = {X 358.1224, Y 47.0454, Z -8.0000, A 0.000, B 0.000, C 0.000 }
gfCNCPoint6[11509] = {X 356.1891, Y 48.0454, Z -8.0000, A 0.000, B 0.000, C 0.000 }
gfCNCPoint6[11510] = {X 353.9990, Y 48.8628, Z -8.0000, A 0.000, B 0.000, C 0.000 }
gfCNCPoint6[11511] = {X 351.7371, Y 49.4530, Z -8.0000, A 0.000, B 0.000, C 0.000 }
gfCNCPoint6[11512] = {X 349.4268, Y 49.8101, Z -8.0000, A 0.000, B 0.000, C 0.000 }
gfCNCPoint6[11513] = {X 347.0922, Y 49.9303, Z -8.0000, A 0.000, B 0.000, C 0.000 }
gfCNCPoint6[11514] = {X 345.0325, Y 49.8956, Z -8.0000, A 0.000, B 0.000, C 0.000 }
gfCNCPoint6[11515] = {X 342.9836, Y 49.6824, Z -8.0000, A 0.000, B 0.000, C 0.000 }
gfCNCPoint6[11516] = {X 340.9609, Y 49.2923, Z -8.0000, A 0.000, B 0.000, C 0.000 }
gfCNCPoint6[11517] = {X 338.9796, Y 48.7283, Z -8.0000, A 0.000, B 0.000, C 0.000 }
gfCNCPoint6[11518] = {X 337.0547, Y 47.9945, Z -8.0000, A 0.000, B 0.000, C 0.000 }
gfCNCPoint6[11519] = {X 335.2007, Y 47.0966, Z -8.0000, A 0.000, B 0.000, C 0.000 }
gfCNCPoint6[11520] = {X 333.6120, Y 46.1150, Z -8.0000, A 0.000, B 0.000, C 0.000 }
gfCNCPoint6[11521] = {X 332.1053, Y 45.0117, Z -8.0000, A 0.000, B 0.000, C 0.000 }
gfCNCPoint6[11522] = {X 330.6899, Y 43.7933, Z -8.0000, A 0.000, B 0.000, C 0.000 }
gfCNCPoint6[11523] = {X 329.7572, Y 43.7998, Z -8.0000, A 0.000, B 0.000, C 0.000 }
gfCNCPoint6[11524] = {X 328.8457, Y 43.6022, Z -8.0000, A 0.000, B 0.000, C 0.000 }
gfCNCPoint6[11525] = {X 327.9994, Y 43.2101, Z -8.0000, A 0.000, B 0.000, C 0.000 }
gfCNCPoint6[11526] = {X 327.2594, Y 42.6425, Z -8.0000, A 0.000, B 0.000, C 0.000 }
gfCNCPoint6[11527] = {X 326.6366, Y 42.0352, Z -8.0000, A 0.000, B 0.000, C 0.000 }
gfCNCPoint6[11528] = {X 326.0198, Y 41.2760, Z -8.0000, A 0.000, B 0.000, C 0.000 }
gfCNCPoint6[11529] = {X 325.5934, Y 40.3956, Z -8.0000, A 0.000, B 0.000, C 0.000 }
gfCNCPoint6[11530] = {X 325.3802, Y 39.4410, Z -8.0000, A 0.000, B 0.000, C 0.000 }
gfCNCPoint6[11531] = {X 325.3913, Y 38.4628, Z -8.0000, A 0.000, B 0.000, C 0.000 }
gfCNCPoint6[11532] = {X 325.6264, Y 37.5133, Z -8.0000, A 0.000, B 0.000, C 0.000 }
gfCNCPoint6[11533] = {X 326.0727, Y 36.6429, Z -8.0000, A 0.000, B 0.000, C 0.000 }
gfCNCPoint6[11534] = {X 330.3061, Y 30.3131, Z -8.0000, A 0.000, B 0.000, C 0.000 }
gfCNCPoint6[11535] = {X 330.8963, Y 29.6095, Z -8.0000, A 0.000, B 0.000, C 0.000 }
gfCNCPoint6[11536] = {X 331.6242, Y 29.0495, Z -8.0000, A 0.000, B 0.000, C 0.000 }
gfCNCPoint6[11537] = {X 332.4556, Y 28.6594, Z -8.0000, A 0.000, B 0.000, C 0.000 }
gfCNCPoint6[11538] = {X 333.3516, Y 28.4575, Z -8.0000, A 0.000, B 0.000, C 0.000 }
gfCNCPoint6[11539] = {X 334.2699, Y 28.4532, Z -8.0000, A 0.000, B 0.000, C 0.000 }
gfCNCPoint6[11540] = {X 335.1677, Y 28.6467, Z -8.0000, A 0.000, B 0.000, C 0.000 }
gfCNCPoint6[11541] = {X 336.0027, Y 29.0291, Z -8.0000, A 0.000, B 0.000, C 0.000 }
gfCNCPoint6[11542] = {X 336.7358, Y 29.5823, Z -8.0000, A 0.000, B 0.000, C 0.000 }
gfCNCPoint6[11543] = {X 337.3723, Y 30.1953, Z -8.0000, A 0.000, B 0.000, C 0.000 }
gfCNCPoint6[11544] = {X 337.9877, Y 30.9588, Z -8.0000, A 0.000, B 0.000, C 0.000 }
gfCNCPoint6[11545] = {X 338.4111, Y 31.8432, Z -8.0000, A 0.000, B 0.000, C 0.000 }
gfCNCPoint6[11546] = {X 338.6201, Y 32.8013, Z -8.0000, A 0.000, B 0.000, C 0.000 }
gfCNCPoint6[11547] = {X 338.6034, Y 33.7818, Z -8.0000, A 0.000, B 0.000, C 0.000 }
gfCNCPoint6[11548] = {X 338.6293, Y 33.9138, Z -8.0000, A 0.000, B 0.000, C 0.000 }
gfCNCPoint6[11549] = {X 339.4398, Y 34.6549, Z -8.0000, A 0.000, B 0.000, C 0.000 }
gfCNCPoint6[11550] = {X 340.5849, Y 35.5676, Z -8.0000, A 0.000, B 0.000, C 0.000 }
gfCNCPoint6[11551] = {X 341.8432, Y 36.3164, Z -8.0000, A 0.000, B 0.000, C 0.000 }
gfCNCPoint6[11552] = {X 343.1915, Y 36.8876, Z -8.0000, A 0.000, B 0.000, C 0.000 }
gfCNCPoint6[11553] = {X 344.6048, Y 37.2705, Z -8.0000, A 0.000, B 0.000, C 0.000 }
gfCNCPoint6[11554] = {X 346.0570, Y 37.4580, Z -8.0000, A 0.000, B 0.000, C 0.000 }
gfCNCPoint6[11555] = {X 347.5213, Y 37.4467, Z -8.0000, A 0.000, B 0.000, C 0.000 }
gfCNCPoint6[11556] = {X 348.6872, Y 37.3098, Z -8.0000, A 0.000, B 0.000, C 0.000 }
gfCNCPoint6[11557] = {X 349.8252, Y 37.0218, Z -8.0000, A 0.000, B 0.000, C 0.000 }
gfCNCPoint6[11558] = {X 350.9159, Y 36.5877, Z -8.0000, A 0.000, B 0.000, C 0.000 }
gfCNCPoint6[11559] = {X 351.9406, Y 36.0149, Z -8.0000, A 0.000, B 0.000, C 0.000 }
gfCNCPoint6[11560] = {X 352.8818, Y 35.3133, Z -8.0000, A 0.000, B 0.000, C 0.000 }
gfCNCPoint6[11561] = {X 354.0422, Y 34.1855, Z -8.0000, A 0.000, B 0.000, C 0.000 }
gfCNCPoint6[11562] = {X 355.0465, Y 32.9166, Z -8.0000, A 0.000, B 0.000, C 0.000 }
gfCNCPoint6[11563] = {X 355.8776, Y 31.5281, Z -8.0000, A 0.000, B 0.000, C 0.000 }
gfCNCPoint6[11564] = {X 356.5214, Y 30.0434, Z -8.0000, A 0.000, B 0.000, C 0.000 }
gfCNCPoint6[11565] = {X 356.9670, Y 28.4878, Z -8.0000, A 0.000, B 0.000, C 0.000 }
gfCNCPoint6[11566] = {X 357.2415, Y 26.7920, Z -8.0000, A 0.000, B 0.000, C 0.000 }
gfCNCPoint6[11567] = {X 357.3534, Y 25.0778, Z -8.0000, A 0.000, B 0.000, C 0.000 }
gfCNCPoint6[11568] = {X 357.3015, Y 23.3607, Z -8.0000, A 0.000, B 0.000, C 0.000 }
gfCNCPoint6[11569] = {X 357.0863, Y 21.6563, Z -8.0000, A 0.000, B 0.000, C 0.000 }
gfCNCPoint6[11570] = {X 356.7303, Y 20.1306, Z -8.0000, A 0.000, B 0.000, C 0.000 }
gfCNCPoint6[11571] = {X 356.1772, Y 18.6648, Z -8.0000, A 0.000, B 0.000, C 0.000 }
gfCNCPoint6[11572] = {X 355.4365, Y 17.2842, Z -8.0000, A 0.000, B 0.000, C 0.000 }
gfCNCPoint6[11573] = {X 354.5211, Y 16.0127, Z -8.0000, A 0.000, B 0.000, C 0.000 }
gfCNCPoint6[11574] = {X 353.6429, Y 15.0777, Z -8.0000, A 0.000, B 0.000, C 0.000 }
gfCNCPoint6[11575] = {X 352.6435, Y 14.2736, Z -8.0000, A 0.000, B 0.000, C 0.000 }
gfCNCPoint6[11576] = {X 351.5422, Y 13.6157, Z -8.0000, A 0.000, B 0.000, C 0.000 }
gfCNCPoint6[11577] = {X 350.3604, Y 13.1169, Z -8.0000, A 0.000, B 0.000, C 0.000 }
gfCNCPoint6[11578] = {X 349.1209, Y 12.7868, Z -8.0000, A 0.000, B 0.000, C 0.000 }
gfCNCPoint6[11579] = {X 347.3424, Y 12.5651, Z -8.0000, A 0.000, B 0.000, C 0.000 }
gfCNCPoint6[11580] = {X 345.5503, Y 12.5820, Z -8.0000, A 0.000, B 0.000, C 0.000 }
gfCNCPoint6[11581] = {X 343.7763, Y 12.8372, Z -8.0000, A 0.000, B 0.000, C 0.000 }
gfCNCPoint6[11582] = {X 342.0521, Y 13.3261, Z -8.0000, A 0.000, B 0.000, C 0.000 }
gfCNCPoint6[11583] = {X 340.4082, Y 14.0401, Z -8.0000, A 0.000, B 0.000, C 0.000 }
gfCNCPoint6[11584] = {X 338.8739, Y 14.9664, Z -8.0000, A 0.000, B 0.000, C 0.000 }
gfCNCPoint6[11585] = {X 338.8431, Y 15.8044, Z -8.0000, A 0.000, B 0.000, C 0.000 }
gfCNCPoint6[11586] = {X 338.6480, Y 16.6198, Z -8.0000, A 0.000, B 0.000, C 0.000 }
gfCNCPoint6[11587] = {X 338.2962, Y 17.3809, Z -8.0000, A 0.000, B 0.000, C 0.000 }
gfCNCPoint6[11588] = {X 337.8015, Y 18.0580, Z -8.0000, A 0.000, B 0.000, C 0.000 }
gfCNCPoint6[11589] = {X 337.1833, Y 18.6244, Z -8.0000, A 0.000, B 0.000, C 0.000 }
gfCNCPoint6[11590] = {X 336.4675, Y 19.1512, Z -8.0000, A 0.000, B 0.000, C 0.000 }
gfCNCPoint6[11591] = {X 335.6668, Y 19.6018, Z -8.0000, A 0.000, B 0.000, C 0.000 }
gfCNCPoint6[11592] = {X 334.7878, Y 19.8694, Z -8.0000, A 0.000, B 0.000, C 0.000 }
gfCNCPoint6[11593] = {X 333.8718, Y 19.9414, Z -8.0000, A 0.000, B 0.000, C 0.000 }
gfCNCPoint6[11594] = {X 332.9618, Y 19.8143, Z -8.0000, A 0.000, B 0.000, C 0.000 }
gfCNCPoint6[11595] = {X 332.1006, Y 19.4942, Z -8.0000, A 0.000, B 0.000, C 0.000 }
gfCNCPoint6[11596] = {X 331.3285, Y 18.9960, Z -8.0000, A 0.000, B 0.000, C 0.000 }
gfCNCPoint6[11597] = {X 330.6819, Y 18.3433, Z -8.0000, A 0.000, B 0.000, C 0.000 }
gfCNCPoint6[11598] = {X 330.1911, Y 17.5665, Z -8.0000, A 0.000, B 0.000, C 0.000 }
gfCNCPoint6[11599] = {X 326.6662, Y 10.3152, Z -8.0000, A 0.000, B 0.000, C 0.000 }
gfCNCPoint6[11600] = {X 326.3374, Y 9.3676, Z -8.0000, A 0.000, B 0.000, C 0.000 }
gfCNCPoint6[11601] = {X 326.2405, Y 8.3693, Z -8.0000, A 0.000, B 0.000, C 0.000 }
gfCNCPoint6[11602] = {X 326.3807, Y 7.3762, Z -8.0000, A 0.000, B 0.000, C 0.000 }
gfCNCPoint6[11603] = {X 326.7504, Y 6.4438, Z -8.0000, A 0.000, B 0.000, C 0.000 }
gfCNCPoint6[11604] = {X 327.3287, Y 5.6243, Z -8.0000, A 0.000, B 0.000, C 0.000 }
gfCNCPoint6[11605] = {X 328.0833, Y 4.9636, Z -8.0000, A 0.000, B 0.000, C 0.000 }
gfCNCPoint6[11606] = {X 328.7533, Y 4.5047, Z -8.0000, A 0.000, B 0.000, C 0.000 }
gfCNCPoint6[11607] = {X 329.6258, Y 4.0538, Z -8.0000, A 0.000, B 0.000, C 0.000 }
gfCNCPoint6[11608] = {X 330.5787, Y 3.8156, Z -8.0000, A 0.000, B 0.000, C 0.000 }
gfCNCPoint6[11609] = {X 331.5608, Y 3.8031, Z -8.0000, A 0.000, B 0.000, C 0.000 }
gfCNCPoint6[11610] = {X 332.5194, Y 4.0169, Z -8.0000, A 0.000, B 0.000, C 0.000 }
gfCNCPoint6[11611] = {X 334.0041, Y 3.1849, Z -8.0000, A 0.000, B 0.000, C 0.000 }
gfCNCPoint6[11612] = {X 335.5370, Y 2.4454, Z -8.0000, A 0.000, B 0.000, C 0.000 }
gfCNCPoint6[11613] = {X 337.6697, Y 1.5776, Z -8.0000, A 0.000, B 0.000, C 0.000 }
gfCNCPoint6[11614] = {X 339.8703, Y 0.9004, Z -8.0000, A 0.000, B 0.000, C 0.000 }
gfCNCPoint6[11615] = {X 342.1218, Y 0.4190, Z -8.0000, A 0.000, B 0.000, C 0.000 }
gfCNCPoint6[11616] = {X 344.4070, Y 0.1371, Z -8.0000, A 0.000, B 0.000, C 0.000 }
gfCNCPoint6[11617] = {X 346.7080, Y 0.0569, Z -8.0000, A 0.000, B 0.000, C 0.000 }
gfCNCPoint6[11618] = {X 349.0072, Y 0.1791, Z -8.0000, A 0.000, B 0.000, C 0.000 }
gfCNCPoint6[11619] = {X 351.2869, Y 0.5026, Z -8.0000, A 0.000, B 0.000, C 0.000 }
gfCNCPoint6[11620] = {X 353.1938, Y 0.9242, Z -8.0000, A 0.000, B 0.000, C 0.000 }
gfCNCPoint6[11621] = {X 355.0531, Y 1.5216, Z -8.0000, A 0.000, B 0.000, C 0.000 }
gfCNCPoint6[11622] = {X 356.8487, Y 2.2896, Z -8.0000, A 0.000, B 0.000, C 0.000 }
gfCNCPoint6[11623] = {X 358.5650, Y 3.2216, Z -8.0000, A 0.000, B 0.000, C 0.000 }
gfCNCPoint6[11624] = {X 360.1870, Y 4.3094, Z -8.0000, A 0.000, B 0.000, C 0.000 }
gfCNCPoint6[11625] = {X 361.7006, Y 5.5435, Z -8.0000, A 0.000, B 0.000, C 0.000 }
gfCNCPoint6[11626] = {X 363.0927, Y 6.9133, Z -8.0000, A 0.000, B 0.000, C 0.000 }
gfCNCPoint6[11627] = {X 364.6348, Y 8.7764, Z -8.0000, A 0.000, B 0.000, C 0.000 }
gfCNCPoint6[11628] = {X 365.9874, Y 10.7814, Z -8.0000, A 0.000, B 0.000, C 0.000 }
gfCNCPoint6[11629] = {X 367.1376, Y 12.9090, Z -8.0000, A 0.000, B 0.000, C 0.000 }
gfCNCPoint6[11630] = {X 368.0742, Y 15.1389, Z -8.0000, A 0.000, B 0.000, C 0.000 }
gfCNCPoint6[11631] = {X 368.7884, Y 17.4496, Z -8.0000, A 0.000, B 0.000, C 0.000 }
gfCNCPoint6[11632] = {X 369.2694, Y 19.7364, Z -8.0000, A 0.000, B 0.000, C 0.000 }
gfCNCPoint6[11633] = {X 369.5796, Y 22.0526, Z -8.0000, A 0.000, B 0.000, C 0.000 }
gfCNCPoint6[11634] = {X 369.7172, Y 24.3855, Z -8.0000, A 0.000, B 0.000, C 0.000 }
gfCNCPoint6[11635] = {X 369.6815, Y 26.7221, Z -8.0000, A 0.000, B 0.000, C 0.000 }
gfCNCPoint6[11636] = {X 369.4727, Y 29.0496, Z -8.0000, A 0.000, B 0.000, C 0.000 }
gfCNCPoint6[11637] = {X 369.0919, Y 31.3553, Z -8.0000, A 0.000, B 0.000, C 0.000 }
gfCNCPoint6[11638] = {X 368.5695, Y 33.4527, Z -8.0000, A 0.000, B 0.000, C 0.000 }
gfCNCPoint6[11639] = {X 367.8639, Y 35.4959, Z -8.0000, A 0.000, B 0.000, C 0.000 }
gfCNCPoint6[11640] = {X 366.9806, Y 37.4687, Z -8.0000, A 0.000, B 0.000, C 0.000 }
gfCNCPoint6[11641] = {X 365.9266, Y 39.3559, Z -8.0000, A 0.000, B 0.000, C 0.000 }
gfCNCPoint6[11642] = {X 364.7101, Y 41.1427, Z -8.0000, A 0.000, B 0.000, C 0.000 }
gfCNCPoint6[11643] = {X 364.6516, Y 41.2226, Z -8.0000, A 0.000, B 0.000, C 0.000 }
gfCNCPoint6[11644] = {X 367.8794, Y 43.5851, Z -8.0000, A 0.000, B 0.000, C 0.000 }
gfCNCPoint6[11645] = {X 364.5871, Y 41.1754, Z -8.0000, A 0.000, B 0.000, C 0.000 }
gfCNCPoint6[11646] = {X 364.5294, Y 41.2541, Z -8.0000, A 0.000, B 0.000, C 0.000 }
gfCNCPoint6[11647] = {X 363.1395, Y 42.9183, Z -8.0000, A 0.000, B 0.000, C 0.000 }
gfCNCPoint6[11648] = {X 361.5913, Y 44.4365, Z -8.0000, A 0.000, B 0.000, C 0.000 }
gfCNCPoint6[11649] = {X 359.9001, Y 45.7935, Z -8.0000, A 0.000, B 0.000, C 0.000 }
gfCNCPoint6[11650] = {X 358.0826, Y 46.9760, Z -8.0000, A 0.000, B 0.000, C 0.000 }
gfCNCPoint6[11651] = {X 356.1567, Y 47.9723, Z -8.0000, A 0.000, B 0.000, C 0.000 }
gfCNCPoint6[11652] = {X 353.9741, Y 48.7867, Z -8.0000, A 0.000, B 0.000, C 0.000 }
gfCNCPoint6[11653] = {X 351.7199, Y 49.3749, Z -8.0000, A 0.000, B 0.000, C 0.000 }
gfCNCPoint6[11654] = {X 349.4176, Y 49.7306, Z -8.0000, A 0.000, B 0.000, C 0.000 }
gfCNCPoint6[11655] = {X 347.0911, Y 49.8503, Z -8.0000, A 0.000, B 0.000, C 0.000 }
gfCNCPoint6[11656] = {X 345.0383, Y 49.8158, Z -8.0000, A 0.000, B 0.000, C 0.000 }
gfCNCPoint6[11657] = {X 342.9962, Y 49.6034, Z -8.0000, A 0.000, B 0.000, C 0.000 }
gfCNCPoint6[11658] = {X 340.9803, Y 49.2147, Z -8.0000, A 0.000, B 0.000, C 0.000 }
gfCNCPoint6[11659] = {X 339.0056, Y 48.6526, Z -8.0000, A 0.000, B 0.000, C 0.000 }
gfCNCPoint6[11660] = {X 337.0872, Y 47.9214, Z -8.0000, A 0.000, B 0.000, C 0.000 }
gfCNCPoint6[11661] = {X 335.2394, Y 47.0266, Z -8.0000, A 0.000, B 0.000, C 0.000 }
gfCNCPoint6[11662] = {X 333.6460, Y 46.0414, Z -8.0000, A 0.000, B 0.000, C 0.000 }
gfCNCPoint6[11663] = {X 332.1354, Y 44.9334, Z -8.0000, A 0.000, B 0.000, C 0.000 }
gfCNCPoint6[11664] = {X 330.7172, Y 43.7094, Z -8.0000, A 0.000, B 0.000, C 0.000 }
gfCNCPoint6[11665] = {X 329.7931, Y 43.7230, Z -8.0000, A 0.000, B 0.000, C 0.000 }
gfCNCPoint6[11666] = {X 328.8887, Y 43.5322, Z -8.0000, A 0.000, B 0.000, C 0.000 }
gfCNCPoint6[11667] = {X 328.0488, Y 43.1464, Z -8.0000, A 0.000, B 0.000, C 0.000 }
gfCNCPoint6[11668] = {X 327.3148, Y 42.5847, Z -8.0000, A 0.000, B 0.000, C 0.000 }
gfCNCPoint6[11669] = {X 326.6925, Y 41.9780, Z -8.0000, A 0.000, B 0.000, C 0.000 }
gfCNCPoint6[11670] = {X 326.0873, Y 41.2331, Z -8.0000, A 0.000, B 0.000, C 0.000 }
gfCNCPoint6[11671] = {X 325.6690, Y 40.3693, Z -8.0000, A 0.000, B 0.000, C 0.000 }
gfCNCPoint6[11672] = {X 325.4597, Y 39.4326, Z -8.0000, A 0.000, B 0.000, C 0.000 }
gfCNCPoint6[11673] = {X 325.4707, Y 38.4730, Z -8.0000, A 0.000, B 0.000, C 0.000 }
gfCNCPoint6[11674] = {X 325.7013, Y 37.5413, Z -8.0000, A 0.000, B 0.000, C 0.000 }
gfCNCPoint6[11675] = {X 326.1392, Y 36.6874, Z -8.0000, A 0.000, B 0.000, C 0.000 }
gfCNCPoint6[11676] = {X 330.3726, Y 30.3576, Z -8.0000, A 0.000, B 0.000, C 0.000 }
gfCNCPoint6[11677] = {X 330.9517, Y 29.6673, Z -8.0000, A 0.000, B 0.000, C 0.000 }
gfCNCPoint6[11678] = {X 331.6659, Y 29.1178, Z -8.0000, A 0.000, B 0.000, C 0.000 }
gfCNCPoint6[11679] = {X 332.4816, Y 28.7351, Z -8.0000, A 0.000, B 0.000, C 0.000 }
gfCNCPoint6[11680] = {X 333.3606, Y 28.5369, Z -8.0000, A 0.000, B 0.000, C 0.000 }
gfCNCPoint6[11681] = {X 334.2617, Y 28.5327, Z -8.0000, A 0.000, B 0.000, C 0.000 }
gfCNCPoint6[11682] = {X 335.1425, Y 28.7227, Z -8.0000, A 0.000, B 0.000, C 0.000 }
gfCNCPoint6[11683] = {X 335.9617, Y 29.0978, Z -8.0000, A 0.000, B 0.000, C 0.000 }
gfCNCPoint6[11684] = {X 336.6810, Y 29.6405, Z -8.0000, A 0.000, B 0.000, C 0.000 }
gfCNCPoint6[11685] = {X 337.3163, Y 30.2523, Z -8.0000, A 0.000, B 0.000, C 0.000 }
gfCNCPoint6[11686] = {X 337.9217, Y 31.0042, Z -8.0000, A 0.000, B 0.000, C 0.000 }
gfCNCPoint6[11687] = {X 338.3376, Y 31.8754, Z -8.0000, A 0.000, B 0.000, C 0.000 }
gfCNCPoint6[11688] = {X 338.5415, Y 32.8190, Z -8.0000, A 0.000, B 0.000, C 0.000 }
gfCNCPoint6[11689] = {X 338.5223, Y 33.7841, Z -8.0000, A 0.000, B 0.000, C 0.000 }
gfCNCPoint6[11690] = {X 338.5558, Y 33.9551, Z -8.0000, A 0.000, B 0.000, C 0.000 }
gfCNCPoint6[11691] = {X 339.3858, Y 34.7139, Z -8.0000, A 0.000, B 0.000, C 0.000 }
gfCNCPoint6[11692] = {X 340.5392, Y 35.6333, Z -8.0000, A 0.000, B 0.000, C 0.000 }
gfCNCPoint6[11693] = {X 341.8067, Y 36.3877, Z -8.0000, A 0.000, B 0.000, C 0.000 }
gfCNCPoint6[11694] = {X 343.1649, Y 36.9631, Z -8.0000, A 0.000, B 0.000, C 0.000 }
gfCNCPoint6[11695] = {X 344.5886, Y 37.3488, Z -8.0000, A 0.000, B 0.000, C 0.000 }
gfCNCPoint6[11696] = {X 346.0514, Y 37.5378, Z -8.0000, A 0.000, B 0.000, C 0.000 }
gfCNCPoint6[11697] = {X 347.5264, Y 37.5266, Z -8.0000, A 0.000, B 0.000, C 0.000 }
gfCNCPoint6[11698] = {X 348.7024, Y 37.3883, Z -8.0000, A 0.000, B 0.000, C 0.000 }
gfCNCPoint6[11699] = {X 349.8504, Y 37.0977, Z -8.0000, A 0.000, B 0.000, C 0.000 }
gfCNCPoint6[11700] = {X 350.9506, Y 36.6598, Z -8.0000, A 0.000, B 0.000, C 0.000 }
gfCNCPoint6[11701] = {X 351.9843, Y 36.0820, Z -8.0000, A 0.000, B 0.000, C 0.000 }
gfCNCPoint6[11702] = {X 352.9337, Y 35.3742, Z -8.0000, A 0.000, B 0.000, C 0.000 }
gfCNCPoint6[11703] = {X 354.1016, Y 34.2391, Z -8.0000, A 0.000, B 0.000, C 0.000 }
gfCNCPoint6[11704] = {X 355.1124, Y 32.9620, Z -8.0000, A 0.000, B 0.000, C 0.000 }
gfCNCPoint6[11705] = {X 355.9488, Y 31.5645, Z -8.0000, A 0.000, B 0.000, C 0.000 }
gfCNCPoint6[11706] = {X 356.5967, Y 30.0703, Z -8.0000, A 0.000, B 0.000, C 0.000 }
gfCNCPoint6[11707] = {X 357.0453, Y 28.5046, Z -8.0000, A 0.000, B 0.000, C 0.000 }
gfCNCPoint6[11708] = {X 357.3210, Y 26.8012, Z -8.0000, A 0.000, B 0.000, C 0.000 }
gfCNCPoint6[11709] = {X 357.4333, Y 25.0793, Z -8.0000, A 0.000, B 0.000, C 0.000 }
gfCNCPoint6[11710] = {X 357.3812, Y 23.3545, Z -8.0000, A 0.000, B 0.000, C 0.000 }
gfCNCPoint6[11711] = {X 357.1652, Y 21.6425, Z -8.0000, A 0.000, B 0.000, C 0.000 }
gfCNCPoint6[11712] = {X 356.8067, Y 20.1068, Z -8.0000, A 0.000, B 0.000, C 0.000 }
gfCNCPoint6[11713] = {X 356.2498, Y 18.6313, Z -8.0000, A 0.000, B 0.000, C 0.000 }
gfCNCPoint6[11714] = {X 355.5042, Y 17.2416, Z -8.0000, A 0.000, B 0.000, C 0.000 }
gfCNCPoint6[11715] = {X 354.5828, Y 15.9618, Z -8.0000, A 0.000, B 0.000, C 0.000 }
gfCNCPoint6[11716] = {X 353.6970, Y 15.0188, Z -8.0000, A 0.000, B 0.000, C 0.000 }
gfCNCPoint6[11717] = {X 352.6890, Y 14.2077, Z -8.0000, A 0.000, B 0.000, C 0.000 }
gfCNCPoint6[11718] = {X 351.5782, Y 13.5443, Z -8.0000, A 0.000, B 0.000, C 0.000 }
gfCNCPoint6[11719] = {X 350.3863, Y 13.0412, Z -8.0000, A 0.000, B 0.000, C 0.000 }
gfCNCPoint6[11720] = {X 349.1360, Y 12.7083, Z -8.0000, A 0.000, B 0.000, C 0.000 }
gfCNCPoint6[11721] = {X 347.5977, Y 12.5020, Z -8.0000, A 0.000, B 0.000, C 0.000 }
gfCNCPoint6[11722] = {X 346.0459, Y 12.4733, Z -8.0000, A 0.000, B 0.000, C 0.000 }
gfCNCPoint6[11723] = {X 344.5010, Y 12.6227, Z -8.0000, A 0.000, B 0.000, C 0.000 }
gfCNCPoint6[11724] = {X 342.9834, Y 12.9482, Z -8.0000, A 0.000, B 0.000, C 0.000 }
gfCNCPoint6[11725] = {X 341.5131, Y 13.4454, Z -8.0000, A 0.000, B 0.000, C 0.000 }
gfCNCPoint6[11726] = {X 340.1095, Y 14.1079, Z -8.0000, A 0.000, B 0.000, C 0.000 }
gfCNCPoint6[11727] = {X 338.7911, Y 14.9268, Z -8.0000, A 0.000, B 0.000, C 0.000 }
gfCNCPoint6[11728] = {X 338.7685, Y 15.7581, Z -8.0000, A 0.000, B 0.000, C 0.000 }
gfCNCPoint6[11729] = {X 338.5811, Y 16.5683, Z -8.0000, A 0.000, B 0.000, C 0.000 }
gfCNCPoint6[11730] = {X 338.2363, Y 17.3249, Z -8.0000, A 0.000, B 0.000, C 0.000 }
gfCNCPoint6[11731] = {X 337.7479, Y 17.9979, Z -8.0000, A 0.000, B 0.000, C 0.000 }
gfCNCPoint6[11732] = {X 337.1353, Y 18.5603, Z -8.0000, A 0.000, B 0.000, C 0.000 }
gfCNCPoint6[11733] = {X 336.4209, Y 19.0861, Z -8.0000, A 0.000, B 0.000, C 0.000 }
gfCNCPoint6[11734] = {X 335.6353, Y 19.5283, Z -8.0000, A 0.000, B 0.000, C 0.000 }
gfCNCPoint6[11735] = {X 334.7729, Y 19.7908, Z -8.0000, A 0.000, B 0.000, C 0.000 }
gfCNCPoint6[11736] = {X 333.8742, Y 19.8614, Z -8.0000, A 0.000, B 0.000, C 0.000 }
gfCNCPoint6[11737] = {X 332.9814, Y 19.7367, Z -8.0000, A 0.000, B 0.000, C 0.000 }
gfCNCPoint6[11738] = {X 332.1364, Y 19.4226, Z -8.0000, A 0.000, B 0.000, C 0.000 }
gfCNCPoint6[11739] = {X 331.3789, Y 18.9339, Z -8.0000, A 0.000, B 0.000, C 0.000 }
gfCNCPoint6[11740] = {X 330.7445, Y 18.2934, Z -8.0000, A 0.000, B 0.000, C 0.000 }
gfCNCPoint6[11741] = {X 330.2630, Y 17.5314, Z -8.0000, A 0.000, B 0.000, C 0.000 }
gfCNCPoint6[11742] = {X 326.7381, Y 10.2803, Z -8.0000, A 0.000, B 0.000, C 0.000 }
gfCNCPoint6[11743] = {X 326.4156, Y 9.3505, Z -8.0000, A 0.000, B 0.000, C 0.000 }
gfCNCPoint6[11744] = {X 326.3205, Y 8.3711, Z -8.0000, A 0.000, B 0.000, C 0.000 }
gfCNCPoint6[11745] = {X 326.4581, Y 7.3967, Z -8.0000, A 0.000, B 0.000, C 0.000 }
gfCNCPoint6[11746] = {X 326.8207, Y 6.4819, Z -8.0000, A 0.000, B 0.000, C 0.000 }
gfCNCPoint6[11747] = {X 327.3881, Y 5.6778, Z -8.0000, A 0.000, B 0.000, C 0.000 }
gfCNCPoint6[11748] = {X 328.1285, Y 5.0296, Z -8.0000, A 0.000, B 0.000, C 0.000 }
gfCNCPoint6[11749] = {X 328.7983, Y 4.5709, Z -8.0000, A 0.000, B 0.000, C 0.000 }
gfCNCPoint6[11750] = {X 329.6630, Y 4.1252, Z -8.0000, A 0.000, B 0.000, C 0.000 }
gfCNCPoint6[11751] = {X 330.6076, Y 3.8926, Z -8.0000, A 0.000, B 0.000, C 0.000 }
gfCNCPoint6[11752] = {X 331.5805, Y 3.8857, Z -8.0000, A 0.000, B 0.000, C 0.000 }
gfCNCPoint6[11753] = {X 332.5283, Y 4.1049, Z -8.0000, A 0.000, B 0.000, C 0.000 }
gfCNCPoint6[11754] = {X 334.0246, Y 3.2645, Z -8.0000, A 0.000, B 0.000, C 0.000 }
gfCNCPoint6[11755] = {X 335.5700, Y 2.5183, Z -8.0000, A 0.000, B 0.000, C 0.000 }
gfCNCPoint6[11756] = {X 337.6962, Y 1.6530, Z -8.0000, A 0.000, B 0.000, C 0.000 }
gfCNCPoint6[11757] = {X 339.8903, Y 0.9778, Z -8.0000, A 0.000, B 0.000, C 0.000 }
gfCNCPoint6[11758] = {X 342.1351, Y 0.4979, Z -8.0000, A 0.000, B 0.000, C 0.000 }
gfCNCPoint6[11759] = {X 344.4134, Y 0.2168, Z -8.0000, A 0.000, B 0.000, C 0.000 }
gfCNCPoint6[11760] = {X 346.7076, Y 0.1369, Z -8.0000, A 0.000, B 0.000, C 0.000 }
gfCNCPoint6[11761] = {X 348.9999, Y 0.2587, Z -8.0000, A 0.000, B 0.000, C 0.000 }
gfCNCPoint6[11762] = {X 351.2727, Y 0.5813, Z -8.0000, A 0.000, B 0.000, C 0.000 }
gfCNCPoint6[11763] = {X 353.1724, Y 1.0013, Z -8.0000, A 0.000, B 0.000, C 0.000 }
gfCNCPoint6[11764] = {X 355.0247, Y 1.5964, Z -8.0000, A 0.000, B 0.000, C 0.000 }
gfCNCPoint6[11765] = {X 356.8136, Y 2.3615, Z -8.0000, A 0.000, B 0.000, C 0.000 }
gfCNCPoint6[11766] = {X 358.5234, Y 3.2899, Z -8.0000, A 0.000, B 0.000, C 0.000 }
gfCNCPoint6[11767] = {X 360.1393, Y 4.3735, Z -8.0000, A 0.000, B 0.000, C 0.000 }
gfCNCPoint6[11768] = {X 361.6471, Y 5.6030, Z -8.0000, A 0.000, B 0.000, C 0.000 }
gfCNCPoint6[11769] = {X 363.0339, Y 6.9676, Z -8.0000, A 0.000, B 0.000, C 0.000 }
gfCNCPoint6[11770] = {X 364.5710, Y 8.8247, Z -8.0000, A 0.000, B 0.000, C 0.000 }
gfCNCPoint6[11771] = {X 365.9192, Y 10.8231, Z -8.0000, A 0.000, B 0.000, C 0.000 }
gfCNCPoint6[11772] = {X 367.0655, Y 12.9437, Z -8.0000, A 0.000, B 0.000, C 0.000 }
gfCNCPoint6[11773] = {X 367.9991, Y 15.1663, Z -8.0000, A 0.000, B 0.000, C 0.000 }
gfCNCPoint6[11774] = {X 368.7109, Y 17.4694, Z -8.0000, A 0.000, B 0.000, C 0.000 }
gfCNCPoint6[11775] = {X 369.1907, Y 19.7504, Z -8.0000, A 0.000, B 0.000, C 0.000 }
gfCNCPoint6[11776] = {X 369.5000, Y 22.0607, Z -8.0000, A 0.000, B 0.000, C 0.000 }
gfCNCPoint6[11777] = {X 369.6372, Y 24.3875, Z -8.0000, A 0.000, B 0.000, C 0.000 }
gfCNCPoint6[11778] = {X 369.6016, Y 26.7181, Z -8.0000, A 0.000, B 0.000, C 0.000 }
gfCNCPoint6[11779] = {X 369.3933, Y 29.0396, Z -8.0000, A 0.000, B 0.000, C 0.000 }
gfCNCPoint6[11780] = {X 369.0135, Y 31.3393, Z -8.0000, A 0.000, B 0.000, C 0.000 }
gfCNCPoint6[11781] = {X 368.4928, Y 33.4300, Z -8.0000, A 0.000, B 0.000, C 0.000 }
gfCNCPoint6[11782] = {X 367.7894, Y 35.4666, Z -8.0000, A 0.000, B 0.000, C 0.000 }
gfCNCPoint6[11783] = {X 366.9090, Y 37.4330, Z -8.0000, A 0.000, B 0.000, C 0.000 }
gfCNCPoint6[11784] = {X 365.8584, Y 39.3141, Z -8.0000, A 0.000, B 0.000, C 0.000 }
gfCNCPoint6[11785] = {X 364.6458, Y 41.0951, Z -8.0000, A 0.000, B 0.000, C 0.000 }
gfCNCPoint6[11786] = {X 364.5871, Y 41.1754, Z -8.0000, A 0.000, B 0.000, C 0.000 }
gfCNCPoint6[11787] = {X 367.8148, Y 43.5379, Z -8.0000, A 0.000, B 0.000, C 0.000 }
gfCNCPoint6[11788] = {X 364.5225, Y 41.1281, Z -8.0000, A 0.000, B 0.000, C 0.000 }
gfCNCPoint6[11789] = {X 364.4652, Y 41.2064, Z -8.0000, A 0.000, B 0.000, C 0.000 }
gfCNCPoint6[11790] = {X 363.0805, Y 42.8643, Z -8.0000, A 0.000, B 0.000, C 0.000 }
gfCNCPoint6[11791] = {X 361.5382, Y 44.3767, Z -8.0000, A 0.000, B 0.000, C 0.000 }
gfCNCPoint6[11792] = {X 359.8534, Y 45.7285, Z -8.0000, A 0.000, B 0.000, C 0.000 }
gfCNCPoint6[11793] = {X 358.0428, Y 46.9066, Z -8.0000, A 0.000, B 0.000, C 0.000 }
gfCNCPoint6[11794] = {X 356.1242, Y 47.8992, Z -8.0000, A 0.000, B 0.000, C 0.000 }
gfCNCPoint6[11795] = {X 353.9491, Y 48.7107, Z -8.0000, A 0.000, B 0.000, C 0.000 }
gfCNCPoint6[11796] = {X 351.7028, Y 49.2967, Z -8.0000, A 0.000, B 0.000, C 0.000 }
gfCNCPoint6[11797] = {X 349.4085, Y 49.6512, Z -8.0000, A 0.000, B 0.000, C 0.000 }
gfCNCPoint6[11798] = {X 347.0900, Y 49.7703, Z -8.0000, A 0.000, B 0.000, C 0.000 }
gfCNCPoint6[11799] = {X 345.0441, Y 49.7360, Z -8.0000, A 0.000, B 0.000, C 0.000 }
gfCNCPoint6[11800] = {X 343.0089, Y 49.5244, Z -8.0000, A 0.000, B 0.000, C 0.000 }
gfCNCPoint6[11801] = {X 340.9997, Y 49.1371, Z -8.0000, A 0.000, B 0.000, C 0.000 }
gfCNCPoint6[11802] = {X 339.0317, Y 48.5770, Z -8.0000, A 0.000, B 0.000, C 0.000 }
gfCNCPoint6[11803] = {X 337.1197, Y 47.8483, Z -8.0000, A 0.000, B 0.000, C 0.000 }
gfCNCPoint6[11804] = {X 335.2780, Y 46.9565, Z -8.0000, A 0.000, B 0.000, C 0.000 }
gfCNCPoint6[11805] = {X 333.6798, Y 45.9678, Z -8.0000, A 0.000, B 0.000, C 0.000 }
gfCNCPoint6[11806] = {X 332.1654, Y 44.8550, Z -8.0000, A 0.000, B 0.000, C 0.000 }
gfCNCPoint6[11807] = {X 330.7443, Y 43.6252, Z -8.0000, A 0.000, B 0.000, C 0.000 }
gfCNCPoint6[11808] = {X 329.8287, Y 43.6460, Z -8.0000, A 0.000, B 0.000, C 0.000 }
gfCNCPoint6[11809] = {X 328.9316, Y 43.4621, Z -8.0000, A 0.000, B 0.000, C 0.000 }
gfCNCPoint6[11810] = {X 328.0980, Y 43.0827, Z -8.0000, A 0.000, B 0.000, C 0.000 }
gfCNCPoint6[11811] = {X 327.3701, Y 42.5270, Z -8.0000, A 0.000, B 0.000, C 0.000 }
gfCNCPoint6[11812] = {X 326.7483, Y 41.9207, Z -8.0000, A 0.000, B 0.000, C 0.000 }
gfCNCPoint6[11813] = {X 326.1548, Y 41.1901, Z -8.0000, A 0.000, B 0.000, C 0.000 }
gfCNCPoint6[11814] = {X 325.7445, Y 40.3430, Z -8.0000, A 0.000, B 0.000, C 0.000 }
gfCNCPoint6[11815] = {X 325.5393, Y 39.4243, Z -8.0000, A 0.000, B 0.000, C 0.000 }
gfCNCPoint6[11816] = {X 325.5500, Y 38.4831, Z -8.0000, A 0.000, B 0.000, C 0.000 }
gfCNCPoint6[11817] = {X 325.7762, Y 37.5694, Z -8.0000, A 0.000, B 0.000, C 0.000 }
gfCNCPoint6[11818] = {X 326.2057, Y 36.7318, Z -8.0000, A 0.000, B 0.000, C 0.000 }
gfCNCPoint6[11819] = {X 330.4391, Y 30.4021, Z -8.0000, A 0.000, B 0.000, C 0.000 }
gfCNCPoint6[11820] = {X 331.0070, Y 29.7251, Z -8.0000, A 0.000, B 0.000, C 0.000 }
gfCNCPoint6[11821] = {X 331.7074, Y 29.1862, Z -8.0000, A 0.000, B 0.000, C 0.000 }
gfCNCPoint6[11822] = {X 332.5074, Y 28.8108, Z -8.0000, A 0.000, B 0.000, C 0.000 }
gfCNCPoint6[11823] = {X 333.3694, Y 28.6165, Z -8.0000, A 0.000, B 0.000, C 0.000 }
gfCNCPoint6[11824] = {X 334.2531, Y 28.6123, Z -8.0000, A 0.000, B 0.000, C 0.000 }
gfCNCPoint6[11825] = {X 335.1169, Y 28.7985, Z -8.0000, A 0.000, B 0.000, C 0.000 }
gfCNCPoint6[11826] = {X 335.9204, Y 29.1663, Z -8.0000, A 0.000, B 0.000, C 0.000 }
gfCNCPoint6[11827] = {X 336.6259, Y 29.6985, Z -8.0000, A 0.000, B 0.000, C 0.000 }
gfCNCPoint6[11828] = {X 337.2602, Y 30.3094, Z -8.0000, A 0.000, B 0.000, C 0.000 }
gfCNCPoint6[11829] = {X 337.8540, Y 31.0468, Z -8.0000, A 0.000, B 0.000, C 0.000 }
gfCNCPoint6[11830] = {X 338.2619, Y 31.9013, Z -8.0000, A 0.000, B 0.000, C 0.000 }
gfCNCPoint6[11831] = {X 338.4618, Y 32.8267, Z -8.0000, A 0.000, B 0.000, C 0.000 }
gfCNCPoint6[11832] = {X 338.4431, Y 33.7733, Z -8.0000, A 0.000, B 0.000, C 0.000 }
gfCNCPoint6[11833] = {X 338.4303, Y 33.8595, Z -8.0000, A 0.000, B 0.000, C 0.000 }
gfCNCPoint6[11834] = {X 338.4158, Y 33.9454, Z -8.0000, A 0.000, B 0.000, C 0.000 }
gfCNCPoint6[11835] = {X 338.5038, Y 34.0159, Z -8.0000, A 0.000, B 0.000, C 0.000 }
gfCNCPoint6[11836] = {X 339.3318, Y 34.7729, Z -8.0000, A 0.000, B 0.000, C 0.000 }
gfCNCPoint6[11837] = {X 340.4936, Y 35.6990, Z -8.0000, A 0.000, B 0.000, C 0.000 }
gfCNCPoint6[11838] = {X 341.7703, Y 36.4589, Z -8.0000, A 0.000, B 0.000, C 0.000 }
gfCNCPoint6[11839] = {X 343.1383, Y 37.0385, Z -8.0000, A 0.000, B 0.000, C 0.000 }
gfCNCPoint6[11840] = {X 344.5723, Y 37.4272, Z -8.0000, A 0.000, B 0.000, C 0.000 }
gfCNCPoint6[11841] = {X 346.0458, Y 37.6176, Z -8.0000, A 0.000, B 0.000, C 0.000 }
gfCNCPoint6[11842] = {X 347.5315, Y 37.6064, Z -8.0000, A 0.000, B 0.000, C 0.000 }
gfCNCPoint6[11843] = {X 348.7177, Y 37.4668, Z -8.0000, A 0.000, B 0.000, C 0.000 }
gfCNCPoint6[11844] = {X 349.8756, Y 37.1736, Z -8.0000, A 0.000, B 0.000, C 0.000 }
gfCNCPoint6[11845] = {X 350.9854, Y 36.7318, Z -8.0000, A 0.000, B 0.000, C 0.000 }
gfCNCPoint6[11846] = {X 352.0279, Y 36.1490, Z -8.0000, A 0.000, B 0.000, C 0.000 }
gfCNCPoint6[11847] = {X 352.9856, Y 35.4351, Z -8.0000, A 0.000, B 0.000, C 0.000 }
gfCNCPoint6[11848] = {X 354.1610, Y 34.2927, Z -8.0000, A 0.000, B 0.000, C 0.000 }
gfCNCPoint6[11849] = {X 355.1782, Y 33.0074, Z -8.0000, A 0.000, B 0.000, C 0.000 }
gfCNCPoint6[11850] = {X 356.0200, Y 31.6009, Z -8.0000, A 0.000, B 0.000, C 0.000 }
gfCNCPoint6[11851] = {X 356.6721, Y 30.0971, Z -8.0000, A 0.000, B 0.000, C 0.000 }
gfCNCPoint6[11852] = {X 357.1235, Y 28.5213, Z -8.0000, A 0.000, B 0.000, C 0.000 }
gfCNCPoint6[11853] = {X 357.4005, Y 26.8104, Z -8.0000, A 0.000, B 0.000, C 0.000 }
gfCNCPoint6[11854] = {X 357.5133, Y 25.0808, Z -8.0000, A 0.000, B 0.000, C 0.000 }
gfCNCPoint6[11855] = {X 357.4610, Y 23.3484, Z -8.0000, A 0.000, B 0.000, C 0.000 }
gfCNCPoint6[11856] = {X 357.2440, Y 21.6288, Z -8.0000, A 0.000, B 0.000, C 0.000 }
gfCNCPoint6[11857] = {X 356.8830, Y 20.0830, Z -8.0000, A 0.000, B 0.000, C 0.000 }
gfCNCPoint6[11858] = {X 356.3225, Y 18.5979, Z -8.0000, A 0.000, B 0.000, C 0.000 }
gfCNCPoint6[11859] = {X 355.5720, Y 17.1991, Z -8.0000, A 0.000, B 0.000, C 0.000 }
gfCNCPoint6[11860] = {X 354.6445, Y 15.9109, Z -8.0000, A 0.000, B 0.000, C 0.000 }
gfCNCPoint6[11861] = {X 353.7511, Y 14.9599, Z -8.0000, A 0.000, B 0.000, C 0.000 }
gfCNCPoint6[11862] = {X 352.7345, Y 14.1419, Z -8.0000, A 0.000, B 0.000, C 0.000 }
gfCNCPoint6[11863] = {X 351.6143, Y 13.4728, Z -8.0000, A 0.000, B 0.000, C 0.000 }
gfCNCPoint6[11864] = {X 350.4121, Y 12.9655, Z -8.0000, A 0.000, B 0.000, C 0.000 }
gfCNCPoint6[11865] = {X 349.1512, Y 12.6297, Z -8.0000, A 0.000, B 0.000, C 0.000 }
gfCNCPoint6[11866] = {X 347.5975, Y 12.4217, Z -8.0000, A 0.000, B 0.000, C 0.000 }
gfCNCPoint6[11867] = {X 346.0301, Y 12.3939, Z -8.0000, A 0.000, B 0.000, C 0.000 }
gfCNCPoint6[11868] = {X 344.4700, Y 12.5466, Z -8.0000, A 0.000, B 0.000, C 0.000 }
gfCNCPoint6[11869] = {X 342.9378, Y 12.8778, Z -8.0000, A 0.000, B 0.000, C 0.000 }
gfCNCPoint6[11870] = {X 341.4538, Y 13.3831, Z -8.0000, A 0.000, B 0.000, C 0.000 }
gfCNCPoint6[11871] = {X 340.0379, Y 14.0558, Z -8.0000, A 0.000, B 0.000, C 0.000 }
gfCNCPoint6[11872] = {X 338.7088, Y 14.8870, Z -8.0000, A 0.000, B 0.000, C 0.000 }
gfCNCPoint6[11873] = {X 338.7152, Y 15.0053, Z -8.0000, A 0.000, B 0.000, C 0.000 }
gfCNCPoint6[11874] = {X 338.6807, Y 15.8056, Z -8.0000, A 0.000, B 0.000, C 0.000 }
gfCNCPoint6[11875] = {X 338.4906, Y 16.5837, Z -8.0000, A 0.000, B 0.000, C 0.000 }
gfCNCPoint6[11876] = {X 338.1521, Y 17.3097, Z -8.0000, A 0.000, B 0.000, C 0.000 }
gfCNCPoint6[11877] = {X 337.6782, Y 17.9555, Z -8.0000, A 0.000, B 0.000, C 0.000 }
gfCNCPoint6[11878] = {X 337.0874, Y 18.4963, Z -8.0000, A 0.000, B 0.000, C 0.000 }
gfCNCPoint6[11879] = {X 336.3744, Y 19.0211, Z -8.0000, A 0.000, B 0.000, C 0.000 }
gfCNCPoint6[11880] = {X 335.6039, Y 19.4547, Z -8.0000, A 0.000, B 0.000, C 0.000 }
gfCNCPoint6[11881] = {X 334.7580, Y 19.7122, Z -8.0000, A 0.000, B 0.000, C 0.000 }
gfCNCPoint6[11882] = {X 333.8766, Y 19.7814, Z -8.0000, A 0.000, B 0.000, C 0.000 }
gfCNCPoint6[11883] = {X 333.0010, Y 19.6592, Z -8.0000, A 0.000, B 0.000, C 0.000 }
gfCNCPoint6[11884] = {X 332.1722, Y 19.3511, Z -8.0000, A 0.000, B 0.000, C 0.000 }
gfCNCPoint6[11885] = {X 331.4293, Y 18.8718, Z -8.0000, A 0.000, B 0.000, C 0.000 }
gfCNCPoint6[11886] = {X 330.8071, Y 18.2436, Z -8.0000, A 0.000, B 0.000, C 0.000 }
gfCNCPoint6[11887] = {X 330.3348, Y 17.4962, Z -8.0000, A 0.000, B 0.000, C 0.000 }
gfCNCPoint6[11888] = {X 326.8101, Y 10.2453, Z -8.0000, A 0.000, B 0.000, C 0.000 }
gfCNCPoint6[11889] = {X 326.4937, Y 9.3334, Z -8.0000, A 0.000, B 0.000, C 0.000 }
gfCNCPoint6[11890] = {X 326.4004, Y 8.3728, Z -8.0000, A 0.000, B 0.000, C 0.000 }
gfCNCPoint6[11891] = {X 326.5354, Y 7.4171, Z -8.0000, A 0.000, B 0.000, C 0.000 }
gfCNCPoint6[11892] = {X 326.8911, Y 6.5199, Z -8.0000, A 0.000, B 0.000, C 0.000 }
gfCNCPoint6[11893] = {X 327.4476, Y 5.7314, Z -8.0000, A 0.000, B 0.000, C 0.000 }
gfCNCPoint6[11894] = {X 328.1737, Y 5.0956, Z -8.0000, A 0.000, B 0.000, C 0.000 }
gfCNCPoint6[11895] = {X 328.8432, Y 4.6371, Z -8.0000, A 0.000, B 0.000, C 0.000 }
gfCNCPoint6[11896] = {X 329.7002, Y 4.1967, Z -8.0000, A 0.000, B 0.000, C 0.000 }
gfCNCPoint6[11897] = {X 330.6365, Y 3.9696, Z -8.0000, A 0.000, B 0.000, C 0.000 }
gfCNCPoint6[11898] = {X 331.6000, Y 3.9684, Z -8.0000, A 0.000, B 0.000, C 0.000 }
gfCNCPoint6[11899] = {X 332.5369, Y 4.1932, Z -8.0000, A 0.000, B 0.000, C 0.000 }
gfCNCPoint6[11900] = {X 334.0448, Y 3.3442, Z -8.0000, A 0.000, B 0.000, C 0.000 }
gfCNCPoint6[11901] = {X 335.6030, Y 2.5912, Z -8.0000, A 0.000, B 0.000, C 0.000 }
gfCNCPoint6[11902] = {X 337.7228, Y 1.7285, Z -8.0000, A 0.000, B 0.000, C 0.000 }
gfCNCPoint6[11903] = {X 339.9103, Y 1.0553, Z -8.0000, A 0.000, B 0.000, C 0.000 }
gfCNCPoint6[11904] = {X 342.1484, Y 0.5767, Z -8.0000, A 0.000, B 0.000, C 0.000 }
gfCNCPoint6[11905] = {X 344.4198, Y 0.2966, Z -8.0000, A 0.000, B 0.000, C 0.000 }
gfCNCPoint6[11906] = {X 346.7071, Y 0.2169, Z -8.0000, A 0.000, B 0.000, C 0.000 }
gfCNCPoint6[11907] = {X 348.9926, Y 0.3384, Z -8.0000, A 0.000, B 0.000, C 0.000 }
gfCNCPoint6[11908] = {X 351.2585, Y 0.6601, Z -8.0000, A 0.000, B 0.000, C 0.000 }
gfCNCPoint6[11909] = {X 353.1510, Y 1.0784, Z -8.0000, A 0.000, B 0.000, C 0.000 }
gfCNCPoint6[11910] = {X 354.9964, Y 1.6712, Z -8.0000, A 0.000, B 0.000, C 0.000 }
gfCNCPoint6[11911] = {X 356.7784, Y 2.4334, Z -8.0000, A 0.000, B 0.000, C 0.000 }
gfCNCPoint6[11912] = {X 358.4818, Y 3.3582, Z -8.0000, A 0.000, B 0.000, C 0.000 }
gfCNCPoint6[11913] = {X 360.0915, Y 4.4377, Z -8.0000, A 0.000, B 0.000, C 0.000 }
gfCNCPoint6[11914] = {X 361.5937, Y 5.6625, Z -8.0000, A 0.000, B 0.000, C 0.000 }
gfCNCPoint6[11915] = {X 362.9752, Y 7.0219, Z -8.0000, A 0.000, B 0.000, C 0.000 }
gfCNCPoint6[11916] = {X 364.5072, Y 8.8729, Z -8.0000, A 0.000, B 0.000, C 0.000 }
gfCNCPoint6[11917] = {X 365.8509, Y 10.8648, Z -8.0000, A 0.000, B 0.000, C 0.000 }
gfCNCPoint6[11918] = {X 366.9935, Y 12.9785, Z -8.0000, A 0.000, B 0.000, C 0.000 }
gfCNCPoint6[11919] = {X 367.9239, Y 15.1937, Z -8.0000, A 0.000, B 0.000, C 0.000 }
gfCNCPoint6[11920] = {X 368.6334, Y 17.4893, Z -8.0000, A 0.000, B 0.000, C 0.000 }
gfCNCPoint6[11921] = {X 369.1119, Y 19.7644, Z -8.0000, A 0.000, B 0.000, C 0.000 }
gfCNCPoint6[11922] = {X 369.4204, Y 22.0687, Z -8.0000, A 0.000, B 0.000, C 0.000 }
gfCNCPoint6[11923] = {X 369.5573, Y 24.3895, Z -8.0000, A 0.000, B 0.000, C 0.000 }
gfCNCPoint6[11924] = {X 369.5217, Y 26.7141, Z -8.0000, A 0.000, B 0.000, C 0.000 }
gfCNCPoint6[11925] = {X 369.3140, Y 29.0296, Z -8.0000, A 0.000, B 0.000, C 0.000 }
gfCNCPoint6[11926] = {X 368.9351, Y 31.3234, Z -8.0000, A 0.000, B 0.000, C 0.000 }
gfCNCPoint6[11927] = {X 368.4161, Y 33.4073, Z -8.0000, A 0.000, B 0.000, C 0.000 }
gfCNCPoint6[11928] = {X 367.7150, Y 35.4372, Z -8.0000, A 0.000, B 0.000, C 0.000 }
gfCNCPoint6[11929] = {X 366.8374, Y 37.3973, Z -8.0000, A 0.000, B 0.000, C 0.000 }
gfCNCPoint6[11930] = {X 365.7902, Y 39.2723, Z -8.0000, A 0.000, B 0.000, C 0.000 }
gfCNCPoint6[11931] = {X 364.5815, Y 41.0475, Z -8.0000, A 0.000, B 0.000, C 0.000 }
gfCNCPoint6[11932] = {X 364.5225, Y 41.1281, Z -8.0000, A 0.000, B 0.000, C 0.000 }
gfCNCPoint6[11933] = {X 367.7503, Y 43.4906, Z -8.0000, A 0.000, B 0.000, C 0.000 }
gfCNCPoint6[11934] = {X 364.4579, Y 41.0809, Z -8.0000, A 0.000, B 0.000, C 0.000 }
gfCNCPoint6[11935] = {X 364.4010, Y 41.1587, Z -8.0000, A 0.000, B 0.000, C 0.000 }
gfCNCPoint6[11936] = {X 363.1253, Y 42.6978, Z -8.0000, A 0.000, B 0.000, C 0.000 }
gfCNCPoint6[11937] = {X 361.7132, Y 44.1128, Z -8.0000, A 0.000, B 0.000, C 0.000 }
gfCNCPoint6[11938] = {X 360.1767, Y 45.3916, Z -8.0000, A 0.000, B 0.000, C 0.000 }
gfCNCPoint6[11939] = {X 358.5288, Y 46.5233, Z -8.0000, A 0.000, B 0.000, C 0.000 }
gfCNCPoint6[11940] = {X 356.7837, Y 47.4984, Z -8.0000, A 0.000, B 0.000, C 0.000 }
gfCNCPoint6[11941] = {X 356.0912, Y 47.8263, Z -8.0000, A 0.000, B 0.000, C 0.000 }
gfCNCPoint6[11942] = {X 353.9238, Y 48.6348, Z -8.0000, A 0.000, B 0.000, C 0.000 }
gfCNCPoint6[11943] = {X 351.6854, Y 49.2187, Z -8.0000, A 0.000, B 0.000, C 0.000 }
gfCNCPoint6[11944] = {X 349.3992, Y 49.5717, Z -8.0000, A 0.000, B 0.000, C 0.000 }
gfCNCPoint6[11945] = {X 347.0889, Y 49.6903, Z -8.0000, A 0.000, B 0.000, C 0.000 }
gfCNCPoint6[11946] = {X 345.0499, Y 49.6562, Z -8.0000, A 0.000, B 0.000, C 0.000 }
gfCNCPoint6[11947] = {X 343.0216, Y 49.4454, Z -8.0000, A 0.000, B 0.000, C 0.000 }
gfCNCPoint6[11948] = {X 341.0192, Y 49.0595, Z -8.0000, A 0.000, B 0.000, C 0.000 }
gfCNCPoint6[11949] = {X 339.0577, Y 48.5013, Z -8.0000, A 0.000, B 0.000, C 0.000 }
gfCNCPoint6[11950] = {X 337.1521, Y 47.7752, Z -8.0000, A 0.000, B 0.000, C 0.000 }
gfCNCPoint6[11951] = {X 335.3167, Y 46.8865, Z -8.0000, A 0.000, B 0.000, C 0.000 }
gfCNCPoint6[11952] = {X 333.7136, Y 45.8940, Z -8.0000, A 0.000, B 0.000, C 0.000 }
gfCNCPoint6[11953] = {X 332.1951, Y 44.7763, Z -8.0000, A 0.000, B 0.000, C 0.000 }
gfCNCPoint6[11954] = {X 330.7711, Y 43.5406, Z -8.0000, A 0.000, B 0.000, C 0.000 }
gfCNCPoint6[11955] = {X 329.8559, Y 43.5681, Z -8.0000, A 0.000, B 0.000, C 0.000 }
gfCNCPoint6[11956] = {X 328.9584, Y 43.3867, Z -8.0000, A 0.000, B 0.000, C 0.000 }
gfCNCPoint6[11957] = {X 328.1256, Y 43.0060, Z -8.0000, A 0.000, B 0.000, C 0.000 }
gfCNCPoint6[11958] = {X 327.4013, Y 42.4458, Z -8.0000, A 0.000, B 0.000, C 0.000 }
gfCNCPoint6[11959] = {X 326.8042, Y 41.8634, Z -8.0000, A 0.000, B 0.000, C 0.000 }
gfCNCPoint6[11960] = {X 326.2223, Y 41.1472, Z -8.0000, A 0.000, B 0.000, C 0.000 }
gfCNCPoint6[11961] = {X 325.8201, Y 40.3166, Z -8.0000, A 0.000, B 0.000, C 0.000 }
gfCNCPoint6[11962] = {X 325.6189, Y 39.4160, Z -8.0000, A 0.000, B 0.000, C 0.000 }
gfCNCPoint6[11963] = {X 325.6294, Y 38.4932, Z -8.0000, A 0.000, B 0.000, C 0.000 }
gfCNCPoint6[11964] = {X 325.8511, Y 37.5974, Z -8.0000, A 0.000, B 0.000, C 0.000 }
gfCNCPoint6[11965] = {X 326.2722, Y 36.7763, Z -8.0000, A 0.000, B 0.000, C 0.000 }
gfCNCPoint6[11966] = {X 330.5290, Y 30.4119, Z -8.0000, A 0.000, B 0.000, C 0.000 }
gfCNCPoint6[11967] = {X 331.0932, Y 29.7536, Z -8.0000, A 0.000, B 0.000, C 0.000 }
gfCNCPoint6[11968] = {X 331.7861, Y 29.2322, Z -8.0000, A 0.000, B 0.000, C 0.000 }
gfCNCPoint6[11969] = {X 332.5750, Y 28.8725, Z -8.0000, A 0.000, B 0.000, C 0.000 }
gfCNCPoint6[11970] = {X 333.4229, Y 28.6911, Z -8.0000, A 0.000, B 0.000, C 0.000 }
gfCNCPoint6[11971] = {X 334.2900, Y 28.6968, Z -8.0000, A 0.000, B 0.000, C 0.000 }
gfCNCPoint6[11972] = {X 335.1355, Y 28.8892, Z -8.0000, A 0.000, B 0.000, C 0.000 }
gfCNCPoint6[11973] = {X 335.9196, Y 29.2593, Z -8.0000, A 0.000, B 0.000, C 0.000 }
gfCNCPoint6[11974] = {X 336.6056, Y 29.7896, Z -8.0000, A 0.000, B 0.000, C 0.000 }
gfCNCPoint6[11975] = {X 337.2041, Y 30.3665, Z -8.0000, A 0.000, B 0.000, C 0.000 }
gfCNCPoint6[11976] = {X 337.7863, Y 31.0894, Z -8.0000, A 0.000, B 0.000, C 0.000 }
gfCNCPoint6[11977] = {X 338.1862, Y 31.9271, Z -8.0000, A 0.000, B 0.000, C 0.000 }
gfCNCPoint6[11978] = {X 338.3822, Y 32.8344, Z -8.0000, A 0.000, B 0.000, C 0.000 }
gfCNCPoint6[11979] = {X 338.3638, Y 33.7624, Z -8.0000, A 0.000, B 0.000, C 0.000 }
gfCNCPoint6[11980] = {X 338.3475, Y 33.8704, Z -8.0000, A 0.000, B 0.000, C 0.000 }
gfCNCPoint6[11981] = {X 338.3283, Y 33.9779, Z -8.0000, A 0.000, B 0.000, C 0.000 }
gfCNCPoint6[11982] = {X 338.4902, Y 34.1119, Z -8.0000, A 0.000, B 0.000, C 0.000 }
gfCNCPoint6[11983] = {X 339.2778, Y 34.8320, Z -8.0000, A 0.000, B 0.000, C 0.000 }
gfCNCPoint6[11984] = {X 340.4119, Y 35.7390, Z -8.0000, A 0.000, B 0.000, C 0.000 }
gfCNCPoint6[11985] = {X 341.6555, Y 36.4887, Z -8.0000, A 0.000, B 0.000, C 0.000 }
gfCNCPoint6[11986] = {X 342.9870, Y 37.0682, Z -8.0000, A 0.000, B 0.000, C 0.000 }
gfCNCPoint6[11987] = {X 344.3832, Y 37.4673, Z -8.0000, A 0.000, B 0.000, C 0.000 }
gfCNCPoint6[11988] = {X 345.8198, Y 37.6792, Z -8.0000, A 0.000, B 0.000, C 0.000 }
gfCNCPoint6[11989] = {X 347.2718, Y 37.7000, Z -8.0000, A 0.000, B 0.000, C 0.000 }
gfCNCPoint6[11990] = {X 347.5356, Y 37.6863, Z -8.0000, A 0.000, B 0.000, C 0.000 }
gfCNCPoint6[11991] = {X 348.7322, Y 37.5455, Z -8.0000, A 0.000, B 0.000, C 0.000 }
gfCNCPoint6[11992] = {X 349.9003, Y 37.2497, Z -8.0000, A 0.000, B 0.000, C 0.000 }
gfCNCPoint6[11993] = {X 351.0197, Y 36.8041, Z -8.0000, A 0.000, B 0.000, C 0.000 }
gfCNCPoint6[11994] = {X 352.0715, Y 36.2161, Z -8.0000, A 0.000, B 0.000, C 0.000 }
gfCNCPoint6[11995] = {X 353.0375, Y 35.4960, Z -8.0000, A 0.000, B 0.000, C 0.000 }
gfCNCPoint6[11996] = {X 354.2204, Y 34.3463, Z -8.0000, A 0.000, B 0.000, C 0.000 }
gfCNCPoint6[11997] = {X 355.2441, Y 33.0528, Z -8.0000, A 0.000, B 0.000, C 0.000 }
gfCNCPoint6[11998] = {X 356.0912, Y 31.6374, Z -8.0000, A 0.000, B 0.000, C 0.000 }
gfCNCPoint6[11999] = {X 356.7475, Y 30.1239, Z -8.0000, A 0.000, B 0.000, C 0.000 }
gfCNCPoint6[12000] = {X 357.2017, Y 28.5381, Z -8.0000, A 0.000, B 0.000, C 0.000 }
gfCNCPoint6[12001] = {X 357.4800, Y 26.8196, Z -8.0000, A 0.000, B 0.000, C 0.000 }
gfCNCPoint6[12002] = {X 357.5933, Y 25.0823, Z -8.0000, A 0.000, B 0.000, C 0.000 }
gfCNCPoint6[12003] = {X 357.5408, Y 23.3422, Z -8.0000, A 0.000, B 0.000, C 0.000 }
gfCNCPoint6[12004] = {X 357.3228, Y 21.6150, Z -8.0000, A 0.000, B 0.000, C 0.000 }
gfCNCPoint6[12005] = {X 356.9594, Y 20.0591, Z -8.0000, A 0.000, B 0.000, C 0.000 }
gfCNCPoint6[12006] = {X 356.3952, Y 18.5644, Z -8.0000, A 0.000, B 0.000, C 0.000 }
gfCNCPoint6[12007] = {X 355.6398, Y 17.1566, Z -8.0000, A 0.000, B 0.000, C 0.000 }
gfCNCPoint6[12008] = {X 354.7062, Y 15.8600, Z -8.0000, A 0.000, B 0.000, C 0.000 }
gfCNCPoint6[12009] = {X 353.8052, Y 14.9010, Z -8.0000, A 0.000, B 0.000, C 0.000 }
gfCNCPoint6[12010] = {X 352.7800, Y 14.0761, Z -8.0000, A 0.000, B 0.000, C 0.000 }
gfCNCPoint6[12011] = {X 351.6503, Y 13.4014, Z -8.0000, A 0.000, B 0.000, C 0.000 }
gfCNCPoint6[12012] = {X 350.4379, Y 12.8898, Z -8.0000, A 0.000, B 0.000, C 0.000 }
gfCNCPoint6[12013] = {X 349.1664, Y 12.5512, Z -8.0000, A 0.000, B 0.000, C 0.000 }
gfCNCPoint6[12014] = {X 347.3712, Y 12.3264, Z -8.0000, A 0.000, B 0.000, C 0.000 }
gfCNCPoint6[12015] = {X 345.5620, Y 12.3405, Z -8.0000, A 0.000, B 0.000, C 0.000 }
gfCNCPoint6[12016] = {X 343.7706, Y 12.5931, Z -8.0000, A 0.000, B 0.000, C 0.000 }
gfCNCPoint6[12017] = {X 342.0281, Y 13.0800, Z -8.0000, A 0.000, B 0.000, C 0.000 }
gfCNCPoint6[12018] = {X 340.3651, Y 13.7925, Z -8.0000, A 0.000, B 0.000, C 0.000 }
gfCNCPoint6[12019] = {X 338.8107, Y 14.7182, Z -8.0000, A 0.000, B 0.000, C 0.000 }
gfCNCPoint6[12020] = {X 338.7183, Y 14.7824, Z -8.0000, A 0.000, B 0.000, C 0.000 }
gfCNCPoint6[12021] = {X 338.6265, Y 14.8473, Z -8.0000, A 0.000, B 0.000, C 0.000 }
gfCNCPoint6[12022] = {X 338.6380, Y 15.0643, Z -8.0000, A 0.000, B 0.000, C 0.000 }
gfCNCPoint6[12023] = {X 338.5595, Y 16.0364, Z -8.0000, A 0.000, B 0.000, C 0.000 }
gfCNCPoint6[12024] = {X 338.2481, Y 16.9606, Z -8.0000, A 0.000, B 0.000, C 0.000 }
gfCNCPoint6[12025] = {X 337.7222, Y 17.7820, Z -8.0000, A 0.000, B 0.000, C 0.000 }
gfCNCPoint6[12026] = {X 337.0133, Y 18.4517, Z -8.0000, A 0.000, B 0.000, C 0.000 }
gfCNCPoint6[12027] = {X 336.3278, Y 18.9560, Z -8.0000, A 0.000, B 0.000, C 0.000 }
gfCNCPoint6[12028] = {X 335.5713, Y 19.3817, Z -8.0000, A 0.000, B 0.000, C 0.000 }
gfCNCPoint6[12029] = {X 334.7407, Y 19.6341, Z -8.0000, A 0.000, B 0.000, C 0.000 }
gfCNCPoint6[12030] = {X 333.8753, Y 19.7014, Z -8.0000, A 0.000, B 0.000, C 0.000 }
gfCNCPoint6[12031] = {X 333.0157, Y 19.5804, Z -8.0000, A 0.000, B 0.000, C 0.000 }
gfCNCPoint6[12032] = {X 332.2025, Y 19.2768, Z -8.0000, A 0.000, B 0.000, C 0.000 }
gfCNCPoint6[12033] = {X 331.4739, Y 18.8049, Z -8.0000, A 0.000, B 0.000, C 0.000 }
gfCNCPoint6[12034] = {X 330.8643, Y 18.1870, Z -8.0000, A 0.000, B 0.000, C 0.000 }
gfCNCPoint6[12035] = {X 330.4023, Y 17.4521, Z -8.0000, A 0.000, B 0.000, C 0.000 }
gfCNCPoint6[12036] = {X 326.8820, Y 10.2103, Z -8.0000, A 0.000, B 0.000, C 0.000 }
gfCNCPoint6[12037] = {X 326.5719, Y 9.3163, Z -8.0000, A 0.000, B 0.000, C 0.000 }
gfCNCPoint6[12038] = {X 326.4804, Y 8.3746, Z -8.0000, A 0.000, B 0.000, C 0.000 }
gfCNCPoint6[12039] = {X 326.6127, Y 7.4376, Z -8.0000, A 0.000, B 0.000, C 0.000 }
gfCNCPoint6[12040] = {X 326.9614, Y 6.5580, Z -8.0000, A 0.000, B 0.000, C 0.000 }
gfCNCPoint6[12041] = {X 327.5070, Y 5.7849, Z -8.0000, A 0.000, B 0.000, C 0.000 }
gfCNCPoint6[12042] = {X 328.2189, Y 5.1616, Z -8.0000, A 0.000, B 0.000, C 0.000 }
gfCNCPoint6[12043] = {X 328.8880, Y 4.7034, Z -8.0000, A 0.000, B 0.000, C 0.000 }
gfCNCPoint6[12044] = {X 329.7043, Y 4.2813, Z -8.0000, A 0.000, B 0.000, C 0.000 }
gfCNCPoint6[12045] = {X 330.5954, Y 4.0567, Z -8.0000, A 0.000, B 0.000, C 0.000 }
gfCNCPoint6[12046] = {X 331.5142, Y 4.0413, Z -8.0000, A 0.000, B 0.000, C 0.000 }
gfCNCPoint6[12047] = {X 332.4122, Y 4.2361, Z -8.0000, A 0.000, B 0.000, C 0.000 }
gfCNCPoint6[12048] = {X 332.5467, Y 4.2807, Z -8.0000, A 0.000, B 0.000, C 0.000 }
gfCNCPoint6[12049] = {X 332.6250, Y 4.2334, Z -8.0000, A 0.000, B 0.000, C 0.000 }
gfCNCPoint6[12050] = {X 332.7035, Y 4.1864, Z -8.0000, A 0.000, B 0.000, C 0.000 }
gfCNCPoint6[12051] = {X 334.1467, Y 3.3813, Z -8.0000, A 0.000, B 0.000, C 0.000 }
gfCNCPoint6[12052] = {X 335.6355, Y 2.6642, Z -8.0000, A 0.000, B 0.000, C 0.000 }
gfCNCPoint6[12053] = {X 336.0092, Y 2.4979, Z -8.0000, A 0.000, B 0.000, C 0.000 }
gfCNCPoint6[12054] = {X 338.0805, Y 1.6898, Z -8.0000, A 0.000, B 0.000, C 0.000 }
gfCNCPoint6[12055] = {X 340.2133, Y 1.0619, Z -8.0000, A 0.000, B 0.000, C 0.000 }
gfCNCPoint6[12056] = {X 342.3920, Y 0.6189, Z -8.0000, A 0.000, B 0.000, C 0.000 }
gfCNCPoint6[12057] = {X 344.6007, Y 0.3638, Z -8.0000, A 0.000, B 0.000, C 0.000 }
gfCNCPoint6[12058] = {X 346.8231, Y 0.2987, Z -8.0000, A 0.000, B 0.000, C 0.000 }
gfCNCPoint6[12059] = {X 349.0429, Y 0.4240, Z -8.0000, A 0.000, B 0.000, C 0.000 }
gfCNCPoint6[12060] = {X 351.2438, Y 0.7387, Z -8.0000, A 0.000, B 0.000, C 0.000 }
gfCNCPoint6[12061] = {X 351.8104, Y 0.8454, Z -8.0000, A 0.000, B 0.000, C 0.000 }
gfCNCPoint6[12062] = {X 353.8994, Y 1.3805, Z -8.0000, A 0.000, B 0.000, C 0.000 }
gfCNCPoint6[12063] = {X 355.9214, Y 2.1300, Z -8.0000, A 0.000, B 0.000, C 0.000 }
gfCNCPoint6[12064] = {X 357.8545, Y 3.0857, Z -8.0000, A 0.000, B 0.000, C 0.000 }
gfCNCPoint6[12065] = {X 359.6776, Y 4.2373, Z -8.0000, A 0.000, B 0.000, C 0.000 }
gfCNCPoint6[12066] = {X 361.3711, Y 5.5723, Z -8.0000, A 0.000, B 0.000, C 0.000 }
gfCNCPoint6[12067] = {X 362.9165, Y 7.0763, Z -8.0000, A 0.000, B 0.000, C 0.000 }
